# B&R Automation Studio project TD52 (part 66)

```c
    /* End of Switch: '<Root>/GasStop8' */
  }

  for (i = 0; i < 7; i++) {
    Gen2_ref_Y->out.rKengMap_P[i] = (real32_T)Gen2_ref_DWork->y_map_i[i];
  }

  Gen2_ref_Y->out.rPos_CBV2 = (real32_T)rtb_Switch_g[6];
  Gen2_ref_Y->out.rPos_CBV3 = (real32_T)rtb_Switch_g[7];
  Gen2_ref_Y->out.bAirAssistIntake = false;
  Gen2_ref_Y->out.bAirAssistExhaust = false;
  Gen2_ref_Y->out.rPos_AAV_Intake = 0.0F;
  Gen2_ref_Y->out.rPos_AAV_Exhaust = 0.0F;
  Gen2_ref_Y->out.TJ_GasO[0] = false;
  Gen2_ref_Y->out.TJ_GasO[3] = false;
  Gen2_ref_Y->out.TJ_GasO[4] = false;
  Gen2_ref_Y->out.TJ_GasM[0] = false;
  Gen2_ref_Y->out.TJ_GasM[1] = ((rtb_SumofElements -
    Gen2_ref_DWork->UnitDelay_DSTATE_dk > rtb_Gain7) &&
    (Gen2_ref_DWork->UnitDelay2_DSTATE_k - Gen2_ref_DWork->UnitDelay1_DSTATE_b >
     Gen2_ref_DWork->UnitDelay3_DSTATE_m) &&
    Gen2_ref_B->BusInput3.fdc.bActive_GasFlowStepLimit);
  Gen2_ref_Y->out.TJ_GasM[2] = ((rtb_SumofElements_l -
    Gen2_ref_DWork->UnitDelay_DSTATE_m > rtb_Sum_gb) &&
    (Gen2_ref_DWork->UnitDelay2_DSTATE_p - Gen2_ref_DWork->UnitDelay1_DSTATE_c2 >
     Gen2_ref_DWork->UnitDelay3_DSTATE_h) &&
    Gen2_ref_B->BusInput3.fdc.bActive_GasFlowStepLimit);
  Gen2_ref_Y->out.TJ_GasM[3] = false;
  Gen2_ref_Y->out.TJ_GasM[4] = false;
  Gen2_ref_Y->out.bSS = Gen2_ref_B->TON2.LogicalOperator3;

  /* Switch: '<S856>/Switch' incorporates:
   *  Constant: '<S856>/Constant2'
   *  RelationalOperator: '<S856>/Relational Operator'
   */
  if (2.2204460492503131E-16 >= rtb_Divide2_f) {
    r = 2.2204460492503131E-16;
  }

  /* End of Switch: '<S856>/Switch' */

  /* BusCreator: '<S16>/Bus Creator' incorporates:
   *  DataTypeConversion: '<S16>/Data Type Conversion20'
   *  Outport: '<Root>/out'
   *  Product: '<S13>/Product'
   */
  Gen2_ref_Y->out.rLHV_est = (real32_T)(rtb_Switch_n / r);

  /* Gain: '<S7>/W2kW' */
  r = 0.001 * rtb_Switch2_g3;

  /* BusCreator: '<Root>/Bus Creator' incorporates:
   *  BusCreator: '<S7>/Bus Creator2'
   *  DataTypeConversion: '<S7>/Data Type Conversion2'
   *  Outport: '<Root>/dbg'
   */
  Gen2_ref_Y->dbg.HLC.Gen2DbgHlcTraj.rP_Set_Delta_FSM = (real32_T)r;

  /* BusCreator generated from: '<S5>/Bus Creator' incorporates:
   *  Constant: '<S307>/Constant2'
   *  DataTypeConversion: '<S272>/Data Type Conversion'
   *  DataTypeConversion: '<S272>/Data Type Conversion1'
   *  DataTypeConversion: '<S272>/Data Type Conversion2'
   *  DataTypeConversion: '<S272>/Data Type Conversion3'
   *  DataTypeConversion: '<S272>/Data Type Conversion4'
   *  DataTypeConversion: '<S272>/Data Type Conversion5'
   *  DataTypeConversion: '<S272>/Data Type Conversion6'
   *  DataTypeConversion: '<S272>/Data Type Conversion7'
   *  DataTypeConversion: '<S272>/Data Type Conversion8'
   *  DataTypeConversion: '<S272>/Data Type Conversion9'
   *  DiscreteIntegrator: '<S307>/Discrete-Time Integrator'
   *  Sum: '<S307>/Sum4'
   */
  Gen2_ref_Y->dbg.FDC.dbgFDC_Filtering.p2s_raw = (real32_T)rtb_p2s;
  Gen2_ref_Y->dbg.FDC.dbgFDC_Filtering.p2s_1stOrd = (real32_T)
    Gen2_ref_B->sf_FILTERnodelay5.y;
  Gen2_ref_Y->dbg.FDC.dbgFDC_Filtering.p2s_2ndOrd = (real32_T)
    Gen2_ref_B->undOrderFilter3.Switch;
  Gen2_ref_Y->dbg.FDC.dbgFDC_Filtering.ne_raw = (real32_T)
    rtb_DataTypeConversion15;
  Gen2_ref_Y->dbg.FDC.dbgFDC_Filtering.ne_1stOrd = (real32_T)
    Gen2_ref_B->sf_FILTERnodelay4.y;
  Gen2_ref_Y->dbg.FDC.dbgFDC_Filtering.ne_2ndOrd = (real32_T)rtb_Switch_kr;
  Gen2_ref_Y->dbg.FDC.dbgFDC_Filtering.p2s_in = (real32_T)rtb_Switch4_p;
  Gen2_ref_Y->dbg.FDC.dbgFDC_Filtering.ne_in = (real32_T)rtb_Switch5_nn;
  Gen2_ref_Y->dbg.FDC.dbgFDC_Filtering.Ratio1stOrd = (real32_T)(1.0 -
    Gen2_ref_DWork->DiscreteTimeIntegrator_DSTATE_d);
  Gen2_ref_Y->dbg.FDC.dbgFDC_Filtering.Ratio2ndOrd = (real32_T)
    Gen2_ref_DWork->DiscreteTimeIntegrator_DSTATE_d;

  /* BusCreator generated from: '<S5>/Bus Creator' incorporates:
   *  DataTypeConversion: '<S5>/Data Type Conversion1'
   *  DataTypeConversion: '<S5>/Data Type Conversion10'
   *  DataTypeConversion: '<S5>/Data Type Conversion11'
   *  DataTypeConversion: '<S5>/Data Type Conversion2'
   *  DataTypeConversion: '<S5>/Data Type Conversion3'
   *  DataTypeConversion: '<S5>/Data Type Conversion4'
   *  DataTypeConversion: '<S5>/Data Type Conversion9'
   *  Product: '<S267>/Divide3'
   */
  Gen2_ref_Y->dbg.FDC.dbgFDC_GasArt1and2.mdot_dyn = (real32_T)rtb_Divide1_h4;
  Gen2_ref_Y->dbg.FDC.dbgFDC_GasArt1and2.mdot_set = (real32_T)rtb_SumofElements;
  Gen2_ref_Y->dbg.FDC.dbgFDC_GasArt1and2.mdot_ss = (real32_T)rtb_Product3_g;
  Gen2_ref_Y->dbg.FDC.dbgFDC_GasArt1and2.rFactCompLR = (real32_T)rtb_Switch2_l;
  Gen2_ref_Y->dbg.FDC.dbgFDC_GasArt1and2.Rgas12 = (real32_T)rtb_Divide3_n_tmp;
  Gen2_ref_Y->dbg.FDC.dbgFDC_GasArt1and2.rdpdt[0] = (real32_T)
    rtb_Switch2_gd_idx_0;
  Gen2_ref_Y->dbg.FDC.dbgFDC_GasArt1and2.rmdot_mix_dyn[0] = (real32_T)R_2inp[0];

  /* BusCreator generated from: '<S5>/Bus Creator' incorporates:
   *  DataTypeConversion: '<S5>/Data Type Conversion5'
   */
  Gen2_ref_Y->dbg.FDC.dbgFDC_GasArt3.rmdot_mix_dyn_M[0] = (real32_T)
    rtb_Divide_ab[0];

  /* BusCreator generated from: '<S5>/Bus Creator' incorporates:
   *  DataTypeConversion: '<S5>/Data Type Conversion1'
   *  DataTypeConversion: '<S5>/Data Type Conversion10'
   */
  Gen2_ref_Y->dbg.FDC.dbgFDC_GasArt1and2.rdpdt[1] = (real32_T)
    rtb_Switch2_gd_idx_1;
  Gen2_ref_Y->dbg.FDC.dbgFDC_GasArt1and2.rmdot_mix_dyn[1] = (real32_T)R_2inp[1];

  /* BusCreator generated from: '<S5>/Bus Creator' incorporates:
   *  DataTypeConversion: '<S5>/Data Type Conversion5'
   */
  Gen2_ref_Y->dbg.FDC.dbgFDC_GasArt3.rmdot_mix_dyn_M[1] = (real32_T)
    rtb_Divide_ab[1];

  /* BusCreator generated from: '<S5>/Bus Creator' incorporates:
   *  DataTypeConversion: '<S5>/Data Type Conversion1'
   *  DataTypeConversion: '<S5>/Data Type Conversion10'
   */
  Gen2_ref_Y->dbg.FDC.dbgFDC_GasArt1and2.rdpdt[2] = (real32_T)
    rtb_Switch2_gd_idx_2;
  Gen2_ref_Y->dbg.FDC.dbgFDC_GasArt1and2.rmdot_mix_dyn[2] = (real32_T)R_2inp[2];

  /* BusCreator generated from: '<S5>/Bus Creator' incorporates:
   *  DataTypeConversion: '<S5>/Data Type Conversion5'
   */
  Gen2_ref_Y->dbg.FDC.dbgFDC_GasArt3.rmdot_mix_dyn_M[2] = (real32_T)
    rtb_Divide_ab[2];

  /* BusCreator generated from: '<S5>/Bus Creator' incorporates:
   *  DataTypeConversion: '<S5>/Data Type Conversion1'
   *  DataTypeConversion: '<S5>/Data Type Conversion10'
   */
  Gen2_ref_Y->dbg.FDC.dbgFDC_GasArt1and2.rdpdt[3] = (real32_T)
    rtb_Switch2_gd_idx_3;
  Gen2_ref_Y->dbg.FDC.dbgFDC_GasArt1and2.rmdot_mix_dyn[3] = (real32_T)R_2inp[3];

  /* BusCreator generated from: '<S5>/Bus Creator' incorporates:
   *  DataTypeConversion: '<S5>/Data Type Conversion12'
   *  DataTypeConversion: '<S5>/Data Type Conversion5'
   *  DataTypeConversion: '<S5>/Data Type Conversion6'
   *  DataTypeConversion: '<S5>/Data Type Conversion7'
   *  DataTypeConversion: '<S5>/Data Type Conversion8'
   *  Product: '<S268>/Divide3'
   */
  Gen2_ref_Y->dbg.FDC.dbgFDC_GasArt3.rmdot_mix_dyn_M[3] = (real32_T)
    rtb_Divide_ab[3];
  Gen2_ref_Y->dbg.FDC.dbgFDC_GasArt3.mdot_dyn_M = (real32_T)rtb_Sum_mf;
  Gen2_ref_Y->dbg.FDC.dbgFDC_GasArt3.mdot_set_M = (real32_T)rtb_SumofElements_l;
  Gen2_ref_Y->dbg.FDC.dbgFDC_GasArt3.mdot_ss_M = (real32_T)rtb_Sum2_a1;
  Gen2_ref_Y->dbg.FDC.dbgFDC_GasArt3.Rgas3 = (real32_T)rtb_Switch_ks;

  /* BusCreator: '<S9>/Bus Creator' incorporates:
   *  DataTypeConversion: '<S9>/Data Type Conversion3'
   */
  Gen2_ref_Y->dbg.ITC.IT_off_start = 0.0F;
  Gen2_ref_Y->dbg.ITC.IT_off_island34 = 0.0F;
  Gen2_ref_Y->dbg.ITC.IT_off_island6 = (real32_T)rtb_Sum1_dh;

  /* BusCreator: '<S19>/Bus Creator' incorporates:
   *  DataTypeConversion: '<S19>/Data Type Conversion2'
   *  DataTypeConversion: '<S19>/Data Type Conversion3'
   *  DataTypeConversion: '<S19>/Data Type Conversion4'
   *  DataTypeConversion: '<S19>/Data Type Conversion5'
   */
  Gen2_ref_Y->dbg.SkipF.NskipPow = (real32_T)rtb_MinMax_n;
  Gen2_ref_Y->dbg.SkipF.NskipMax = (real32_T)rtb_RoundingFunction;
  Gen2_ref_Y->dbg.SkipF.Nskip34 = (real32_T)rtb_Product1_mqz;
  Gen2_ref_Y->dbg.SkipF.Nskip6 = (real32_T)rtb_Switch2_d1;

  /* Logic: '<S14>/Logical Operator2' */
  Gen2_ref_Y->dbg.LamLim.bInitLamOffs = !rtb_LogicalOperator5_mv;

  /* BusCreator: '<S14>/Bus Creator' incorporates:
   *  DataTypeConversion: '<S14>/Data Type Conversion'
   *  DataTypeConversion: '<S14>/Data Type Conversion10'
   *  DataTypeConversion: '<S14>/Data Type Conversion2'
   *  DataTypeConversion: '<S14>/Data Type Conversion3'
   *  DataTypeConversion: '<S14>/Data Type Conversion4'
   *  DataTypeConversion: '<S14>/Data Type Conversion5'
   *  DataTypeConversion: '<S14>/Data Type Conversion7'
   *  DataTypeConversion: '<S14>/Data Type Conversion8'
   *  DataTypeConversion: '<S14>/Data Type Conversion9'
   *  DataTypeConversion: '<S4>/Data Type Conversion28'
   */
  Gen2_ref_Y->dbg.LamLim.extOffset = Gen2_ref_B->BusInput.rOffsetLamLimit;
  Gen2_ref_Y->dbg.LamLim.AutoOffset = (real32_T)Gen2_ref_B->Filter_l.Switch;
  Gen2_ref_Y->dbg.LamLim.ScaledOffsetUpLim = (real32_T)rtb_Product1_b;
  Gen2_ref_Y->dbg.LamLim.ScaledOffsetLoLim = (real32_T)rtb_Product_l0;
  Gen2_ref_Y->dbg.LamLim.offsetUpLim = (real32_T)rtb_Sum5_j;
  Gen2_ref_Y->dbg.LamLim.offsetLoLim = (real32_T)rtb_Sum8_m;
  Gen2_ref_Y->dbg.LamLim.LamLoLim = (real32_T)rtb_Switch1_k;
  Gen2_ref_Y->dbg.LamLim.LamUpLim = (real32_T)rtb_Switch2_n5;
  Gen2_ref_Y->dbg.LamLim.LamSteadyState = (real32_T)rtb_PactOut_o;
  Gen2_ref_Y->dbg.LamLim.rLamOffsInit = (real32_T)rtb_Divide6_n;
  Gen2_ref_Y->dbg.LamLim.bPminSSadaptReached_Hys = rtb_LogicalOperator12_a;

  /* Gain: '<Root>/W2kW' */
  rtb_Sum8_m = 0.001 * rtb_Gain2_ao;

  /* S-Function (sfix_look1_dyn): '<S865>/LCRScal_CD1' */
  /* Dynamic Look-Up Table Block: '<S865>/LCRScal_CD1'
   * Input0  Data Type:  Floating Point real_T
   * Input1  Data Type:  Floating Point real_T
   * Input2  Data Type:  Floating Point real_T
   * Output0 Data Type:  Floating Point real_T
   * Lookup Method: Linear_Endpoint
   *
   */
  LookUp_real_T_real_T( &(rtb_CDSet_50),
                       &Gen2_ref_B->BusInput3.bdcWgv.rCd_vect_y[0],
                       Gen2_ref_B->BusInput3.leanox.rWG_1,
                       &Gen2_ref_B->BusInput3.bdcWgv.rCd_vect_x[0], 10U, inst);

  /* S-Function (sfix_look1_dyn): '<S865>/LCRScal_CD2' */
  /* Dynamic Look-Up Table Block: '<S865>/LCRScal_CD2'
   * Input0  Data Type:  Floating Point real_T
   * Input1  Data Type:  Floating Point real_T
   * Input2  Data Type:  Floating Point real_T
   * Output0 Data Type:  Floating Point real_T
   * Lookup Method: Linear_Endpoint
   *
   */
  LookUp_real_T_real_T( &(rtb_CDSet_100),
                       &Gen2_ref_B->BusInput3.bdcWgv.rCd_vect_y[0],
                       Gen2_ref_B->BusInput3.leanox.rWG_2,
                       &Gen2_ref_B->BusInput3.bdcWgv.rCd_vect_x[0], 10U, inst);

  /* SignalConversion generated from: '<S867>/ SFunction ' incorporates:
   *  MATLAB Function: '<S15>/LookUp Extrapolation'
   *  SignalConversion generated from: '<S15>/LCRScal_DPWG4'
   */
  rtb_TmpSignalConversionAtLoo_ht[0] = Gen2_ref_B->BusInput3.leanox.rP_1;
  rtb_TmpSignalConversionAtLoo_ht[1] = Gen2_ref_B->BusInput3.leanox.rP_2;

  /* SignalConversion generated from: '<S867>/ SFunction ' incorporates:
   *  MATLAB Function: '<S15>/LookUp Extrapolation'
   */
  rtb_TmpSignalConversionAtLook_d[0] = rtb_CDSet_50;
  rtb_TmpSignalConversionAtLook_d[1] = rtb_CDSet_100;

  /* MATLAB Function: '<S15>/LookUp Extrapolation' */
  if (rtb_TmpSignalConversionAtLoo_ht[0] == rtb_TmpSignalConversionAtLoo_ht[1])
  {
    rtb_DataTypeConversion15 = 0.0;
  } else {
    rtb_DataTypeConversion15 = (rtb_TmpSignalConversionAtLook_d[1] -
      rtb_TmpSignalConversionAtLook_d[0]) / (rtb_TmpSignalConversionAtLoo_ht[1]
      - rtb_TmpSignalConversionAtLoo_ht[0]);
    rtb_DataTypeConversion15 = (rtb_TmpSignalConversionAtLook_d[0] -
      rtb_TmpSignalConversionAtLoo_ht[0] * rtb_DataTypeConversion15) +
      rtb_DataTypeConversion15 * rtb_Sum8_m;
    if (!(rtb_DataTypeConversion15 >= 0.0)) {
      rtb_DataTypeConversion15 = 0.0;
    }

    if (!(rtb_DataTypeConversion15 <= 1.0)) {
      rtb_DataTypeConversion15 = 1.0;
    }
  }

  /* DataTypeConversion: '<S15>/Data Type Conversion' */
  r = Gen2_ref_B->BusInput.tLvrt.rWgPosFb;

  /* Gain: '<S15>/Gain' */
  rtb_Sum_e = 100.0 * r;

  /* S-Function (sfix_look1_dyn): '<S15>/LCRScal_DPWG2' */
  /* Dynamic Look-Up Table Block: '<S15>/LCRScal_DPWG2'
   * Input0  Data Type:  Floating Point real_T
   * Input1  Data Type:  Floating Point real_T
   * Input2  Data Type:  Floating Point real_T
   * Output0 Data Type:  Floating Point real_T
   * Lookup Method: Linear_Endpoint
   *
   */
  LookUp_real_T_real_T( &(rtb_Sum_mf), &Gen2_ref_B->BusInput3.bdcWgv.rCd_vect_y
                       [0], rtb_Sum_e, &Gen2_ref_B->BusInput3.bdcWgv.rCd_vect_x
                       [0], 10U, inst);

  /* BusCreator: '<Root>/Bus Creator1' incorporates:
   *  DataTypeConversion: '<Root>/Data Type Conversion4'
   */
  Gen2_ref_Y->dbg.LxWgvCmp.CDAct = (real32_T)rtb_Sum_mf;

  /* Math: '<S868>/Math Function' */
  r = Gen2_ref_B->BusInput3.bdcWgv.rDref * Gen2_ref_B->BusInput3.bdcWgv.rDref;

  /* Abs: '<S871>/Abs' */
  rtb_Divide2_f = fabs(Gen2_ref_B->BusInput3.eng.rVol_Hub_Eng);

  /* Switch: '<S871>/Switch' incorporates:
   *  Constant: '<S871>/Constant2'
   *  RelationalOperator: '<S871>/Relational Operator'
   */
  if (2.2204460492503131E-16 >= rtb_Divide2_f) {
    rtb_Divide2_f = 2.2204460492503131E-16;
  } else {
    rtb_Divide2_f = Gen2_ref_B->BusInput3.eng.rVol_Hub_Eng;
  }

  /* End of Switch: '<S871>/Switch' */

  /* Product: '<S868>/Divide' incorporates:
   *  Constant: '<S868>/Constant'
   *  Sum: '<S15>/Add1'
   */
  rtb_Sum_mf = (rtb_DataTypeConversion15 - rtb_Sum_mf) * r * 0.78539816339744828
    * Gen2_ref_B->BusInput3.eng.rNum_WGV / rtb_Divide2_f;

  /* SignalConversion generated from: '<S15>/LCRScal_DPWG4' */
  rtb_TmpSignalConversionAtLook_d[0] = rtb_TmpSignalConversionAtLoo_ht[0];
  rtb_TmpSignalConversionAtLook_d[1] = rtb_TmpSignalConversionAtLoo_ht[1];

  /* S-Function (sfix_look1_dyn): '<S15>/LCRScal_DPWG3' */
  /* Dynamic Look-Up Table Block: '<S15>/LCRScal_DPWG3'
   * Input0  Data Type:  Floating Point real_T
   * Input1  Data Type:  Floating Point real_T
   * Input2  Data Type:  Floating Point real_T
   * Output0 Data Type:  Floating Point real_T
   * Lookup Method: Linear_Endpoint
   *
   */
  LookUp_real_T_real_T( &(r), &Gen2_ref_B->BusInput3.leanox.Comp_WG_1_y[0],
                       rtb_Sum_mf, &Gen2_ref_B->BusInput3.leanox.Comp_WG_1_x[0],
                       9U, inst);

  /* S-Function (sfix_look1_dyn): '<S15>/LCRScal_DPWG1' */
  /* Dynamic Look-Up Table Block: '<S15>/LCRScal_DPWG1'
   * Input0  Data Type:  Floating Point real_T
   * Input1  Data Type:  Floating Point real_T
   * Input2  Data Type:  Floating Point real_T
   * Output0 Data Type:  Floating Point real_T
   * Lookup Method: Linear_Endpoint
   *
   */
  LookUp_real_T_real_T( &(rtb_Divide2_f),
                       &Gen2_ref_B->BusInput3.leanox.Comp_WG_2_y[0], rtb_Sum_mf,
                       &Gen2_ref_B->BusInput3.leanox.Comp_WG_2_x[0], 9U, inst);

  /* SignalConversion generated from: '<S15>/LCRScal_DPWG4' */
  rtb_TmpSignalConversionAtLoo_ht[0] = r;
  rtb_TmpSignalConversionAtLoo_ht[1] = rtb_Divide2_f;

  /* S-Function (sfix_look1_dyn): '<S15>/LCRScal_DPWG4' */
  /* Dynamic Look-Up Table Block: '<S15>/LCRScal_DPWG4'
   * Input0  Data Type:  Floating Point real_T
   * Input1  Data Type:  Floating Point real_T
   * Input2  Data Type:  Floating Point real_T
   * Output0 Data Type:  Floating Point real_T
   * Lookup Method: Linear_Endpoint
   *
   */
  LookUp_real_T_real_T( &(r), &rtb_TmpSignalConversionAtLoo_ht[0], rtb_Sum8_m,
                       &rtb_TmpSignalConversionAtLook_d[0], 1U, inst);

  /* BusCreator: '<Root>/Bus Creator1' incorporates:
   *  DataTypeConversion: '<Root>/Data Type Conversion3'
   *  DataTypeConversion: '<Root>/Data Type Conversion5'
   *  DataTypeConversion: '<Root>/Data Type Conversion6'
   *  DataTypeConversion: '<Root>/Data Type Conversion8'
   *  Delay: '<S15>/Resettable Delay'
   */
  Gen2_ref_Y->dbg.LxWgvCmp.CDSet = (real32_T)rtb_DataTypeConversion15;
  Gen2_ref_Y->dbg.LxWgvCmp.DeltaCD_aux = (real32_T)rtb_Sum_mf;
  Gen2_ref_Y->dbg.LxWgvCmp.DeltaP2s_set = (real32_T)r;
  Gen2_ref_Y->dbg.LxWgvCmp.DeltaP2s_Comp_WGV = (real32_T)
    Gen2_ref_DWork->ResettableDelay_DSTATE;

  /* BusCreator: '<S6>/Bus Creator' incorporates:
   *  Delay: '<Root>/Delay6'
   */
  Gen2_ref_Y->dbg.GQC.bActGasQualImprov = rtb_bActGasQualImprov;
  Gen2_ref_Y->dbg.GQC.bDetSatLambda = rtb_LogicalOperator2_fy;
  Gen2_ref_Y->dbg.GQC.bDetKnock = rtb_Switch2_jv;
  Gen2_ref_Y->dbg.GQC.bDetSatActuators = Gen2_ref_DWork->Delay6_DSTATE;
  Gen2_ref_Y->dbg.GQC.bMisfDet = rtb_Switch4_mu;

  /* BusCreator: '<Root>/Bus Creator' incorporates:
   *  BusCreator: '<S427>/Bus Creator5'
   *  BusCreator: '<S429>/Bus Creator'
   *  DataTypeConversion: '<S418>/Data Type Conversion10'
   *  DataTypeConversion: '<S418>/Data Type Conversion11'
   *  DataTypeConversion: '<S418>/Data Type Conversion12'
   *  DataTypeConversion: '<S418>/Data Type Conversion13'
   *  DataTypeConversion: '<S427>/Data Type Conversion'
   *  DataTypeConversion: '<S427>/Data Type Conversion1'
   *  DataTypeConversion: '<S427>/Data Type Conversion2'
   *  DataTypeConversion: '<S427>/Data Type Conversion3'
   *  DataTypeConversion: '<S427>/Data Type Conversion4'
   *  DataTypeConversion: '<S429>/Data Type Conversion1'
   *  DataTypeConversion: '<S429>/Data Type Conversion4'
   *  DataTypeConversion: '<S429>/Data Type Conversion5'
   *  DataTypeConversion: '<S432>/Data Type Conversion1'
   *  DataTypeConversion: '<S432>/Data Type Conversion10'
   *  DataTypeConversion: '<S432>/Data Type Conversion11'
   *  DataTypeConversion: '<S432>/Data Type Conversion2'
   *  DataTypeConversion: '<S432>/Data Type Conversion3'
   *  DataTypeConversion: '<S432>/Data Type Conversion4'
   *  DataTypeConversion: '<S432>/Data Type Conversion5'
   *  DataTypeConversion: '<S432>/Data Type Conversion6'
   *  DataTypeConversion: '<S581>/Data Type Conversion6'
   *  Outport: '<Root>/dbg'
   *  Quantizer: '<S581>/Quantizer1'
   */
  Gen2_ref_Y->dbg.HLCi.FF.rPest_FF = (real32_T)rtb_Switch_bs;
  Gen2_ref_Y->dbg.HLCi.FF.rP2s_FF = (real32_T)rtb_mbar2pa_g;
  Gen2_ref_Y->dbg.HLCi.FF.P_est_vFilt = (real32_T)rtb_Switch2_gs;
  Gen2_ref_Y->dbg.HLCi.FF.LineVol_nPower = (real32_T)rtb_Switch_iy;
  Gen2_ref_Y->dbg.HLCi.FF.LineVol_vPower = (real32_T)rtb_rKK2_k;
  Gen2_ref_Y->dbg.HLCi.FF.rFactLSL = (real32_T)rtb_Sum1_jz;
  Gen2_ref_Y->dbg.HLCi.FF.rLSLff_p = (real32_T)rtb_Divide_kp;
  Gen2_ref_Y->dbg.HLCi.FF.rLSLff_d = (real32_T)rtb_Divide2_a;
  Gen2_ref_Y->dbg.HLCi.LR.bLR_GasStop = rtb_TOF_IN;
  Gen2_ref_Y->dbg.HLCi.LR.bIgnOff = rtb_bCBV_min;
  Gen2_ref_Y->dbg.HLCi.LR.bLR_ActSat_CBV =
    Gen2_ref_B->TP_ActSat_CBV.LogicalOperator1;
  Gen2_ref_Y->dbg.HLCi.LR.bLR_ActSat_TV =
    Gen2_ref_B->TP_ActSat_TV.LogicalOperator1;
  Gen2_ref_Y->dbg.HLCi.LR.bLR_IGN_Retard_Trig = rtb_RelationalOperator2_j;
  Gen2_ref_Y->dbg.HLCi.LR.rP_Rot_Corr_Norm = (real32_T)rtb_Saturation;
  Gen2_ref_Y->dbg.HLCi.LR.IGN_retard_interpol = (real32_T)rtb_Switch2_jq;
  Gen2_ref_Y->dbg.HLCi.LR.IGN_retard_active = (real32_T)rtb_Divide4_d;
  Gen2_ref_Y->dbg.HLCi.LR.delta_IGN_Retard = (real32_T)rtb_MinMax_a;
  Gen2_ref_Y->dbg.HLCi.LR.rFactCompLR = (real32_T)rtb_Switch2_l;
  Gen2_ref_Y->dbg.HLCi.LR.bLR_SatActuators = rtb_LogicalOperator3_gq;
  Gen2_ref_Y->dbg.HLCi.Prot.omega = (real32_T)rtb_Gain;
  Gen2_ref_Y->dbg.HLCi.Prot.omega_filt = (real32_T)rtb_Switch_eu;
  Gen2_ref_Y->dbg.HLCi.Prot.omega_dot = (real32_T)rtb_Switch1_mm;
  Gen2_ref_Y->dbg.HLCi.Prot.rProt = (real32_T)rtb_Gain1_fr;
  Gen2_ref_Y->dbg.HLCi.SkipF.rSkipfire_PI = (real32_T)rtb_Switch2_ba;
  Gen2_ref_Y->dbg.HLCi.SkipF.rLam_skip = (real32_T)rtb_Switch_fi;
  Gen2_ref_Y->dbg.HLCi.SkipF.bDemand_Skip = rtb_LogicalOperator1_ja;
  Gen2_ref_Y->dbg.HLCi.SkipF.rSkip_level = (real32_T)rtb_rSkip_level;
  Gen2_ref_Y->dbg.HLCi.SkipF.rSkipfire = (real32_T)rtb_Divide1_f1_tmp;
  Gen2_ref_Y->dbg.HLCi.SkipF.bSkip_pulse_on = rtb_LogicalOperator1_pa;

  /* Switch: '<S429>/Switch1' incorporates:
   *  BusCreator: '<Root>/Bus Creator'
   *  DataTypeConversion: '<S429>/Data Type Conversion2'
   *  Outport: '<Root>/dbg'
   */
  Gen2_ref_Y->dbg.HLCi.SkipF.rN_diff = (real32_T)rtb_Divide_mr_tmp;

  /* BusCreator: '<Root>/Bus Creator' incorporates:
   *  BusCreator: '<S1>/Bus Creator2'
   *  BusCreator: '<S23>/Bus Creator1'
   *  BusCreator: '<S389>/Bus Creator1'
   *  BusCreator: '<S431>/Bus Creator'
   *  BusCreator: '<S7>/Bus Creator2'
   *  DataTypeConversion: '<S12>/Data Type Conversion1'
   *  DataTypeConversion: '<S1>/Data Type Conversion'
   *  DataTypeConversion: '<S1>/Data Type Conversion1'
   *  DataTypeConversion: '<S1>/Data Type Conversion10'
   *  DataTypeConversion: '<S1>/Data Type Conversion16'
   *  DataTypeConversion: '<S1>/Data Type Conversion17'
   *  DataTypeConversion: '<S1>/Data Type Conversion18'
   *  DataTypeConversion: '<S1>/Data Type Conversion2'
   *  DataTypeConversion: '<S1>/Data Type Conversion22'
   *  DataTypeConversion: '<S1>/Data Type Conversion23'
   *  DataTypeConversion: '<S1>/Data Type Conversion24'
   *  DataTypeConversion: '<S1>/Data Type Conversion3'
   *  DataTypeConversion: '<S1>/Data Type Conversion4'
   *  DataTypeConversion: '<S1>/Data Type Conversion5'
   *  DataTypeConversion: '<S1>/Data Type Conversion6'
   *  DataTypeConversion: '<S1>/Data Type Conversion8'
   *  DataTypeConversion: '<S23>/Data Type Conversion'
   *  DataTypeConversion: '<S23>/Data Type Conversion1'
   *  DataTypeConversion: '<S23>/Data Type Conversion2'
   *  DataTypeConversion: '<S23>/Data Type Conversion3'
   *  DataTypeConversion: '<S23>/Data Type Conversion4'
   *  DataTypeConversion: '<S23>/Data Type Conversion6'
   *  DataTypeConversion: '<S23>/Data Type Conversion7'
   *  DataTypeConversion: '<S26>/Data Type Conversion'
   *  DataTypeConversion: '<S26>/Data Type Conversion2'
   *  DataTypeConversion: '<S26>/Data Type Conversion3'
   *  DataTypeConversion: '<S26>/Data Type Conversion4'
   *  DataTypeConversion: '<S26>/Data Type Conversion5'
   *  DataTypeConversion: '<S26>/Data Type Conversion7'
   *  DataTypeConversion: '<S379>/Data Type Conversion10'
   *  DataTypeConversion: '<S379>/Data Type Conversion3'
   *  DataTypeConversion: '<S379>/Data Type Conversion5'
   *  DataTypeConversion: '<S379>/Data Type Conversion8'
   *  DataTypeConversion: '<S389>/Data Type Conversion3'
   *  DataTypeConversion: '<S389>/Data Type Conversion6'
   *  DataTypeConversion: '<S389>/Data Type Conversion8'
   *  DataTypeConversion: '<S431>/Data Type Conversion1'
   *  DataTypeConversion: '<S431>/Data Type Conversion10'
   *  DataTypeConversion: '<S431>/Data Type Conversion11'
   *  DataTypeConversion: '<S431>/Data Type Conversion12'
   *  DataTypeConversion: '<S431>/Data Type Conversion13'
   *  DataTypeConversion: '<S431>/Data Type Conversion14'
   *  DataTypeConversion: '<S431>/Data Type Conversion15'
   *  DataTypeConversion: '<S431>/Data Type Conversion16'
   *  DataTypeConversion: '<S431>/Data Type Conversion17'
   *  DataTypeConversion: '<S431>/Data Type Conversion18'
   *  DataTypeConversion: '<S431>/Data Type Conversion19'
   *  DataTypeConversion: '<S431>/Data Type Conversion2'
   *  DataTypeConversion: '<S431>/Data Type Conversion20'
   *  DataTypeConversion: '<S431>/Data Type Conversion21'
   *  DataTypeConversion: '<S431>/Data Type Conversion22'
   *  DataTypeConversion: '<S431>/Data Type Conversion23'
   *  DataTypeConversion: '<S431>/Data Type Conversion24'
   *  DataTypeConversion: '<S431>/Data Type Conversion25'
   *  DataTypeConversion: '<S431>/Data Type Conversion26'
   *  DataTypeConversion: '<S431>/Data Type Conversion27'
   *  DataTypeConversion: '<S431>/Data Type Conversion3'
   *  DataTypeConversion: '<S431>/Data Type Conversion4'
   *  DataTypeConversion: '<S431>/Data Type Conversion5'
   *  DataTypeConversion: '<S431>/Data Type Conversion6'
   *  DataTypeConversion: '<S431>/Data Type Conversion7'
   *  DataTypeConversion: '<S431>/Data Type Conversion8'
   *  DataTypeConversion: '<S431>/Data Type Conversion9'
   *  DataTypeConversion: '<S43>/Data Type Conversion1'
   *  DataTypeConversion: '<S43>/Data Type Conversion24'
   *  DataTypeConversion: '<S43>/Data Type Conversion25'
   *  DataTypeConversion: '<S43>/Data Type Conversion3'
   *  DataTypeConversion: '<S45>/Data Type Conversion'
   *  DataTypeConversion: '<S45>/Data Type Conversion2'
   *  DataTypeConversion: '<S45>/Data Type Conversion3'
   *  DataTypeConversion: '<S45>/Data Type Conversion4'
   *  DataTypeConversion: '<S45>/Data Type Conversion7'
   *  DataTypeConversion: '<S4>/Data Type Conversion29'
   *  DataTypeConversion: '<S78>/Data Type Conversion1'
   *  DataTypeConversion: '<S78>/Data Type Conversion10'
   *  DataTypeConversion: '<S78>/Data Type Conversion2'
   *  DataTypeConversion: '<S78>/Data Type Conversion3'
   *  DataTypeConversion: '<S78>/Data Type Conversion4'
   *  DataTypeConversion: '<S78>/Data Type Conversion5'
   *  DataTypeConversion: '<S78>/Data Type Conversion7'
   *  DataTypeConversion: '<S78>/Data Type Conversion8'
   *  DataTypeConversion: '<S78>/Data Type Conversion9'
   *  DataTypeConversion: '<S7>/Data Type Conversion1'
   *  DiscreteIntegrator: '<S26>/Discrete-Time Integrator'
   *  DiscreteIntegrator: '<S45>/Discrete-Time Integrator1'
   *  DiscreteIntegrator: '<S62>/Discrete-Time Integrator'
   *  DiscreteIntegrator: '<S748>/Discrete-Time Integrator4'
   *  Gain: '<S431>/Gain1'
   *  Gain: '<S7>/Pa2bar'
   *  Logic: '<S45>/Logical Operator'
   *  MATLAB Function: '<S431>/LQR Controller 3states'
   *  Outport: '<Root>/dbg'
   *  SignalConversion generated from: '<S627>/ SFunction '
   *  Sum: '<S641>/Sum2'
   *  Sum: '<S641>/Sum6'
   */
  Gen2_ref_Y->dbg.HLCi.LQR.x_ref[0] = (real32_T)rtb_Saturation6;
  Gen2_ref_Y->dbg.HLCi.LQR.x_ref[1] = (real32_T)rtb_Abs;
  Gen2_ref_Y->dbg.HLCi.LQR.x_ref[2] = (real32_T)rtb_Switch2_c4;
  Gen2_ref_Y->dbg.HLCi.LQR.x_sp[0] = (real32_T)rtb_Sum1_l;
  Gen2_ref_Y->dbg.HLCi.LQR.x_sp[1] = (real32_T)rtb_Sum2_a_tmp;
  Gen2_ref_Y->dbg.HLCi.LQR.x_sp[2] = (real32_T)rtb_Sum6_o_tmp;
  Gen2_ref_Y->dbg.HLCi.LQR.x_k[0] = (real32_T)rtb_Gain1_f_tmp;
  Gen2_ref_Y->dbg.HLCi.LQR.x_k[1] = (real32_T)rtb_Gain3;
  Gen2_ref_Y->dbg.HLCi.LQR.x_k[2] = (real32_T)Gen2_ref_B->Filter_bd.Switch;
  Gen2_ref_Y->dbg.HLCi.LQR.u_k[0] = (real32_T)rtb_Product_m[0];
  Gen2_ref_Y->dbg.HLCi.LQR.u_k[1] = (real32_T)rtb_Product_m[1];
  Gen2_ref_Y->dbg.HLCi.LQR.u_k[2] = (real32_T)rtb_Product_m[2];
  Gen2_ref_Y->dbg.HLCi.LQR.u_k[3] = (real32_T)rtb_Product_m[3];
  Gen2_ref_Y->dbg.HLCi.LQR.x_dist1_map = (real32_T)rtb_Gain1_o;
  Gen2_ref_Y->dbg.HLCi.LQR.x_KF[0] = (real32_T)rtb_x_KF_out_idx_0;
  Gen2_ref_Y->dbg.HLCi.LQR.x_dist_KF[0] = (real32_T)rtb_Switch1_cl[0];
  Gen2_ref_Y->dbg.HLCi.LQR.x_sp_KF[0] = (real32_T)rtb_x_sp_KF_idx_0;
  Gen2_ref_Y->dbg.HLCi.LQR.x_KF[1] = (real32_T)rtb_x_KF_out_idx_1;
  Gen2_ref_Y->dbg.HLCi.LQR.x_dist_KF[1] = (real32_T)rtb_Switch1_cl[1];
  Gen2_ref_Y->dbg.HLCi.LQR.x_sp_KF[1] = (real32_T)rtb_x_sp_KF_idx_1;
  Gen2_ref_Y->dbg.HLCi.LQR.x_KF[2] = (real32_T)rtb_x_KF_out_idx_2;
  Gen2_ref_Y->dbg.HLCi.LQR.x_dist_KF[2] = (real32_T)rtb_Switch1_cl[2];
  Gen2_ref_Y->dbg.HLCi.LQR.x_sp_KF[2] = (real32_T)rtb_x_sp_KF_idx_2;
  Gen2_ref_Y->dbg.HLCi.LQR.u_sp_KF[0] = (real32_T)rtb_u_sp_KF[0];
  Gen2_ref_Y->dbg.HLCi.LQR.u_sp_KF[1] = (real32_T)rtb_u_sp_KF[1];
  Gen2_ref_Y->dbg.HLCi.LQR.err_KF[0] = (real32_T)rtb_err_KF[0];
  Gen2_ref_Y->dbg.HLCi.LQR.err_KF[1] = (real32_T)rtb_err_KF[1];
  Gen2_ref_Y->dbg.HLCi.LQR.err_KF[2] = (real32_T)rtb_err_KF[2];
  for (i = 0; i < 18; i++) {
    Gen2_ref_Y->dbg.HLCi.LQR.K_KF[i] = (real32_T)rtb_K_KF_out[i];
  }

  for (i = 0; i < 36; i++) {
    Gen2_ref_Y->dbg.HLCi.LQR.P_KF[i] = (real32_T)Gen2_ref_DWork->P_KF[i];
  }

  Gen2_ref_Y->dbg.HLCi.LQR.err_cont[0] = (real32_T)rtb_err_cont[0];
  Gen2_ref_Y->dbg.HLCi.LQR.err_cont[1] = (real32_T)rtb_err_cont[1];
  Gen2_ref_Y->dbg.HLCi.LQR.err_cont[2] = (real32_T)rtb_err_cont[2];
  Gen2_ref_Y->dbg.HLCi.LQR.Ke_calc = (real32_T)rtb_Switch_nb;
  Gen2_ref_Y->dbg.HLCi.LQR.Ke = (real32_T)rtb_Product_o;
  Gen2_ref_Y->dbg.HLCi.LQR.Ke0 = (real32_T)rtb_VariableIntegerDelay;
  Gen2_ref_Y->dbg.HLCi.LQR.eOmRef = (real32_T)rtb_Switch_dhr;
  Gen2_ref_Y->dbg.HLCi.LQR.bTrigDPr_limit = rtb_Act;
  Gen2_ref_Y->dbg.HLCi.LQR.bOutOfNWindow = rtb_LogicalOperator4_go;
  Gen2_ref_Y->dbg.HLCi.LQR.omega_dot = (real32_T)((rtb_Product_o / (y_map_tmp_0 *
    rtb_Sum1_idx_2 + 1.0) * y_map_tmp * (rtb_Product_m[2] *
    Gen2_ref_B->BusInput3.SpeedCtrl.rK_it2_iLQR + 1.0) - rtb_Divide_i1) * (1.0 /
    rtb_TmpSignalConversionAtSFunct[3]));
  Gen2_ref_Y->dbg.HLCi.LQR.bLamSat = rtb_LogicalOperator2_ov;
  for (i = 0; i < 9; i++) {
    Gen2_ref_Y->dbg.HLCi.LQR.Phi[i] = (real32_T)rtb_Phi_OUT[i];
  }

  Gen2_ref_Y->dbg.HLCi.LQR.x_k_pred[0] = (real32_T)
    rtb_TmpSignalConversionAtSFun_g[0];
  Gen2_ref_Y->dbg.HLCi.LQR.x_k_pred[1] = (real32_T)
    rtb_TmpSignalConversionAtSFun_g[1];
  Gen2_ref_Y->dbg.HLCi.LQR.x_k_pred[2] = (real32_T)
    rtb_TmpSignalConversionAtSFun_g[2];
  for (i = 0; i < 12; i++) {
    Gen2_ref_Y->dbg.HLCi.LQR.H[i] = (real32_T)rtb_H_OUT[i];
    Gen2_ref_Y->dbg.HLCi.LQR.K_LQR[i] = (real32_T)rtb_K_LQR[i];
  }

  for (i = 0; i < 9; i++) {
    Gen2_ref_Y->dbg.HLCi.LQR.P_LQR[i] = (real32_T)Gen2_ref_DWork->P[i];
  }

  Gen2_ref_Y->dbg.HLCi.LQR.Ke_act_map = (real32_T)rtb_Switch1_ep;
  Gen2_ref_Y->dbg.HLCi.LQR.bAdaptReleased = rtb_RelationalOperator_ok;
  Gen2_ref_Y->dbg.HLCi.LQR.bResKeEst = rtb_Switch2_ij;
  Gen2_ref_Y->dbg.HLCi.LQR.bKeEstTransDet = rtb_Switch3_of;
  Gen2_ref_Y->dbg.HLCi.LQR.Ke_est = (real32_T)Gen2_ref_B->Filter1_o.Switch;
  Gen2_ref_Y->dbg.HLCi.LQR.delta_IT_Acc = (real32_T)rtb_Product4_d;
  Gen2_ref_Y->dbg.HLCi.LQR.dPr_P2s_RefSatLam = (real32_T)
    Gen2_ref_DWork->DiscreteTimeIntegrator4_DSTATE;
  Gen2_ref_Y->dbg.HLC.Gen2DbgHlcTraj.rp2s_leanox = (real32_T)(1.0E-5 *
    rtb_Pa2bar_k);

  /* Outputs for Atomic SubSystem: '<S342>/PID_Power' */
  Gen2_ref_Y->dbg.HLC.BGen2DbgHlcPowCtrl.ff = (real32_T)rtb_Switch_e3;
  Gen2_ref_Y->dbg.HLC.BGen2DbgHlcPowCtrl.ud = (real32_T)rtb_Divide3_p;
  Gen2_ref_Y->dbg.HLC.BGen2DbgHlcPowCtrl.aw_ext = (real32_T)rtb_Switch8;

  /* End of Outputs for SubSystem: '<S342>/PID_Power' */
  Gen2_ref_Y->dbg.HLC.BGen2DbgHlcPowCtrl.aw_aux =
    Gen2_ref_B->BusInput.rAW_EGT_ext;

  /* Outputs for Atomic SubSystem: '<S342>/PID_Power' */
  Gen2_ref_Y->dbg.HLC.BGen2DbgHlcPowCtrl.u = (real32_T)rtb_Switch2_jw;

  /* End of Outputs for SubSystem: '<S342>/PID_Power' */

  /* Outputs for Atomic SubSystem: '<S343>/PID_Power' */
  Gen2_ref_Y->dbg.HLC.dbgHLCPowCtrlGQC.ff = 0.0F;

  /* End of Outputs for SubSystem: '<S343>/PID_Power' */
  Gen2_ref_Y->dbg.HLC.dbgHLCPowCtrlGQC.ui = rtb_BusCreator1_h_ui;

  /* Outputs for Atomic SubSystem: '<S343>/PID_Power' */
  Gen2_ref_Y->dbg.HLC.dbgHLCPowCtrlGQC.ud = (real32_T)rtb_Divide3_d;
  Gen2_ref_Y->dbg.HLC.dbgHLCPowCtrlGQC.aw_ext = 0.0F;
  Gen2_ref_Y->dbg.HLC.dbgHLCPowCtrlGQC.aw_aux = (real32_T)rtb_Product1;
  Gen2_ref_Y->dbg.HLC.dbgHLCPowCtrlGQC.u = (real32_T)
    Gen2_ref_B->sf_MATLABFunction1_ep.LamOut;

  /* End of Outputs for SubSystem: '<S343>/PID_Power' */
  Gen2_ref_Y->dbg.BDC.Misc.PI_tv = (real32_T)rtb_Divide_br;
  Gen2_ref_Y->dbg.BDC.Misc.PI_LP = (real32_T)rtb_Divide2;
  Gen2_ref_Y->dbg.BDC.Misc.PI_HP = (real32_T)rtb_Divide1_fn;
  Gen2_ref_Y->dbg.BDC.Misc.PI_total = (real32_T)rtb_Divide3_a0;
  Gen2_ref_Y->dbg.BDC.tv.ff = (real32_T)
    Gen2_ref_B->Inverse_Linearization1.LCRScal_Lam_EOT1;
  Gen2_ref_Y->dbg.BDC.tv.up = (real32_T)rtb_Product4;
  Gen2_ref_Y->dbg.BDC.tv.ui = (real32_T)
    Gen2_ref_DWork->DiscreteTimeIntegrator1_DSTAT_n;
  Gen2_ref_Y->dbg.BDC.tv.uaw = (real32_T)rtb_Switch2_oou;
  Gen2_ref_Y->dbg.BDC.tv.i0 = (real32_T)rtb_Switch1_d2;
  Gen2_ref_Y->dbg.BDC.tv.bTVCtrl_ON = !rtb_i_reset;
  Gen2_ref_Y->dbg.BDC.cbv.ff_cbv = (real32_T)rtb_Saturation1_i;
  Gen2_ref_Y->dbg.BDC.cbv.ff_cbv_unsat = (real32_T)rtb_Sum1_lo;
  Gen2_ref_Y->dbg.BDC.cbv.up_cbv = (real32_T)rtb_up;
  Gen2_ref_Y->dbg.BDC.cbv.ui_cbv = (real32_T)
    Gen2_ref_DWork->DiscreteTimeIntegrator_DSTAT_ja;
  Gen2_ref_Y->dbg.BDC.cbv.uaw_cbv = (real32_T)FILT_IN;
  Gen2_ref_Y->dbg.BDC.cbv.i0_cbv = (real32_T)rtb_Add2_h;
  Gen2_ref_Y->dbg.BDC.SP.rCBV_Min = (real32_T)rtb_Switch2_a;
  Gen2_ref_Y->dbg.BDC.SP.rTV_Min = (real32_T)rtb_Switch_e;
  Gen2_ref_Y->dbg.BDC.SP.rMdot_mixture_cyl = (real32_T)rtb_MassFlowCalc;
  Gen2_ref_Y->dbg.BDC.SP.rPrR_TC_Surge = (real32_T)rtb_Saturation_gh;
  Gen2_ref_Y->dbg.BDC.MP.u = (real32_T)rtb_Sum11;
  Gen2_ref_Y->dbg.BDC.MP.u_ff = (real32_T)rtb_MinMax1_h;
  Gen2_ref_Y->dbg.BDC.MP.u0 = (real32_T)rtb_Sum7_l5;
  Gen2_ref_Y->dbg.BDC.MP.u0_ff = (real32_T)rtb_MinMax1_g;
  Gen2_ref_Y->dbg.BDC.MP.TVdp = (real32_T)rtb_Product2;
  Gen2_ref_Y->dbg.BDC.MP.offset = (real32_T)
    Gen2_ref_DWork->DiscreteTimeIntegrator_DSTATE_a;
  Gen2_ref_Y->dbg.BDC.MP.offset_in = (real32_T)rtb_Gain_kl;
  Gen2_ref_Y->dbg.BDC.RL.RLp2s_d = (real32_T)rtb_p1LP;
  Gen2_ref_Y->dbg.BDC.RL.RLp2s_d_ff = (real32_T)rtb_p1HP;
  Gen2_ref_Y->dbg.BDC.RL.RLp2s_d_ff_z = (real32_T)rtb_VariableIntegerDelay_b;
  Gen2_ref_Y->dbg.BDC.RL.RLact = (real32_T)rtb_MinMax3;
  Gen2_ref_Y->dbg.BDC.RL.RL = (real32_T)rtb_MinMax_mf;
  Gen2_ref_Y->dbg.BDC.RL.Rlrequ = (real32_T)rtb_Divide_kt;
  Gen2_ref_Y->dbg.BDC.RL.RLp2s_d_RL = (real32_T)rtb_p2HP;
  Gen2_ref_Y->dbg.BDC.RL.RLp2s_d_ff_RL = (real32_T)rtb_Sum5_iu;
  Gen2_ref_Y->dbg.BDC.RL.Rlreset = rtb_LogicalOperator3_ja;
  Gen2_ref_Y->dbg.BDC.traj.ref_P2_FF_CBV = rtb_Switch2_h1;
  Gen2_ref_Y->dbg.BDC.traj.ref_P2s_FF = rtb_Switch2_lu;
  Gen2_ref_Y->dbg.BDC.traj.ref_P2_FF = rtb_BusCreator1_ref_P2_FF;
  Gen2_ref_Y->dbg.BDC.traj.ref_P2s_FB_TV = rtb_BusCreator1_ref_P2s_FB_TV;
  Gen2_ref_Y->dbg.BDC.traj.ref_P2_FB_CBV = rtb_BusCreator1_ref_P2_FB_CBV;
  Gen2_ref_Y->dbg.BDC.traj.ref_P2s_FF_TV = rtb_Switch2_jf;
  Gen2_ref_Y->dbg.BDC.traj.d_dt_ref_P2s_FF_TV = Gen2_ref_B->Filter2.Switch1;
  Gen2_ref_Y->dbg.BDC.traj.d_dt_ref_P2_FF_CBV = Gen2_ref_B->Filter1.Switch1;
  Gen2_ref_Y->dbg.BDC.traj.d_dt_ref_P2s_FF = Gen2_ref_B->Filter4.Switch1;
  Gen2_ref_Y->dbg.BDC.FF.me = (real32_T)rtb_dm_e;
  Gen2_ref_Y->dbg.BDC.FF.me_d = (real32_T)Gen2_ref_B->sf_enginemassflow.dm_e;
  Gen2_ref_Y->dbg.BDC.FF.me_cbv_d = (real32_T)rtb_Abs_n;
  Gen2_ref_Y->dbg.BDC.FF.TV_me_d = (real32_T)rtb_Divide_n0;
  Gen2_ref_Y->dbg.BDC.FF.wg_me = (real32_T)Gen2_ref_B->sf_enginemassflow1_e.dm_e;
  Gen2_ref_Y->dbg.BDC.FF.wg_me_d = (real32_T)
    Gen2_ref_B->sf_enginemassflow_h.dm_e;
  Gen2_ref_Y->dbg.BDC.FF.wg_m_d = (real32_T)rtb_Saturation_cx;
  Gen2_ref_Y->dbg.BDC.FF.u_ff_cbv = (real32_T)rtb_Sum1_lo;
  Gen2_ref_Y->dbg.BDC.FF.dbg_cbvTracking_PI = (real32_T)rtb_Sum3_hx;
  Gen2_ref_Y->dbg.BDC.FF.dbg_cbvTracking_P = (real32_T)rtb_Divide1_k;
  Gen2_ref_Y->dbg.BDC.FF.dbg_cbvTracking_I = (real32_T)
    rtb_DiscreteTimeIntegrator_g3;
  Gen2_ref_Y->dbg.KeEstNetP.KeEstNetP = (real32_T)Gen2_ref_B->Filter1_n.Switch;

  /* S-Function (bur_bus_out): '<Root>/Bus Output' incorporates:
   *  Outport: '<Root>/dbg'
   */
  inst->dbgOut = Gen2_ref_Y->dbg;

  /* S-Function (bur_bus_out): '<Root>/Bus Output1' incorporates:
   *  Outport: '<Root>/out'
   */
  inst->OUT = Gen2_ref_Y->out;

  /* S-Function (bur_in): '<Root>/Input1' */
  Gen2_ref_B->Input1 = inst->rLam_BrakeEffEst;

  /* Outputs for Atomic SubSystem: '<Root>/brake eff estimate' */
  /* Gain: '<S21>/Gain' */
  rtb_Sum_mf = 0.10471975511965977 * Gen2_ref_B->BusInput3.eng.rN_Nom;

  /* Product: '<S21>/Divide' */
  rtb_Sum_mf = Gen2_ref_B->BusInput3.eng.rVol_Hub_Eng * rtb_Sum1_idx_3 *
    rtb_Sum_mf * rtb_etaVolConst_lt * Gen2_ref_B->p2s_filt.Switch;

  /* Product: '<S21>/Divide3' */
  rtb_Divide2_f = Gen2_ref_B->Input1 * rtb_Sum1_idx_2;

  /* Sum: '<S21>/Sum1' incorporates:
   *  Constant: '<S21>/Constant2'
   */
  rtb_Gain = rtb_Divide2_f + 1.0;

  /* Gain: '<S21>/Gain1' */
  rtb_Divide2_f = rtb_Switch2_ejy_tmp;

  /* Saturate: '<S21>/Saturation3' */
  if (rtb_Sum_mf <= 1.0) {
    rtb_Sum_mf = 1.0;
  }

  /* End of Saturate: '<S21>/Saturation3' */

  /* Product: '<S21>/Divide2' incorporates:
   *  Constant: '<S21>/Constant'
   *  Product: '<S21>/Divide1'
   *  Sum: '<S21>/Sum2'
   */
  u0 = rtb_Gain * rtb_kW2W * Gen2_ref_B->T2s_filt.Switch *
    (Gen2_ref_B->Pel_filt.Switch + rtb_Divide2_f) * 12.566370614359172 * (1.0 /
    rtb_Sum_mf);

  /* Saturate: '<S21>/Saturation2' */
  if (u0 > 1.0) {
    /* DataTypeConversion: '<Root>/Data Type Conversion1' */
    Gen2_ref_B->DataTypeConversion1 = 1.0F;
  } else if (u0 < 0.0001) {
    /* DataTypeConversion: '<Root>/Data Type Conversion1' */
    Gen2_ref_B->DataTypeConversion1 = 0.0001F;
  } else {
    /* DataTypeConversion: '<Root>/Data Type Conversion1' */
    Gen2_ref_B->DataTypeConversion1 = (real32_T)u0;
  }

  /* End of Saturate: '<S21>/Saturation2' */
  /* End of Outputs for SubSystem: '<Root>/brake eff estimate' */

  /* S-Function (bur_out): '<Root>/Output' */
  inst->rEtaBrakeEst = Gen2_ref_B->DataTypeConversion1;

  /* DataTypeConversion: '<S22>/Data Type Conversion' incorporates:
   *  Constant: '<S47>/Constant'
   *  DiscreteIntegrator: '<S22>/Discrete-Time Integrator'
   *  RelationalOperator: '<S47>/Compare'
   */
  rtb_Sum_mf = (Gen2_ref_DWork->DiscreteTimeIntegrator_DSTATE_i > 0.0);

  /* Product: '<S22>/Product1' */
  rtb_Divide2_f = rtb_Gain_kp * Gen2_ref_B->BusInput3.bdcWgv.rKiWgvTcOvrspdCtrl;

  /* Product: '<S22>/Product2' */
  rtb_Gain = Gen2_ref_B->BusInput3.bdcWgv.rIntDischargeTcOvrspedCtrl *
    rtb_Sum_mf;

  /* Saturate: '<S22>/Saturation2' */
  if (rtb_Divide2_f <= 0.0) {
    delta_y = 0.0;
  } else {
    delta_y = rtb_Divide2_f;
  }

  /* End of Saturate: '<S22>/Saturation2' */

  /* DataTypeConversion: '<S48>/Data Type Conversion1' incorporates:
   *  Constant: '<S66>/Constant'
   *  DiscreteIntegrator: '<S48>/Discrete-Time Integrator'
   *  RelationalOperator: '<S66>/Compare'
   */
  rtb_Sum_mf = (Gen2_ref_DWork->DiscreteTimeIntegrator_DSTAT_ac > 0.0);

  /* Product: '<S48>/Product3' */
  rtb_Divide2_f = rtb_Divide3_k *
    Gen2_ref_B->BusInput3.bdcMisc.rKiSurgeProtectSL;

  /* Sum: '<S48>/Sum11' incorporates:
   *  Product: '<S48>/Product4'
   */
  rtb_Switch_eu = rtb_Divide2_f -
    Gen2_ref_B->BusInput3.bdcMisc.rIntDischargeSurgeCtrl * rtb_Sum_mf;

  /* Sum: '<S26>/Sum2' incorporates:
   *  MATLAB Function: '<S26>/fb_err'
   *  Product: '<S26>/Product1'
   */
  rtb_Switch1_mm = err * rtb_Pa2bar + FILT_IN;

  /* Saturate: '<S132>/Saturation' */
  if (Gen2_ref_B->BusInput3.bdcMisc.rTiF_Pr_p2s > 1000.0) {
    FILT_IN = 1000.0;
  } else if (Gen2_ref_B->BusInput3.bdcMisc.rTiF_Pr_p2s < 0.001) {
    FILT_IN = 0.001;
  } else {
    FILT_IN = Gen2_ref_B->BusInput3.bdcMisc.rTiF_Pr_p2s;
  }

  /* End of Saturate: '<S132>/Saturation' */

  /* Product: '<S132>/Divide' incorporates:
   *  DiscreteIntegrator: '<S132>/Discrete-Time Integrator'
   *  Sum: '<S132>/Sum4'
   */
  rtb_Gain1_fr = (Gen2_ref_B->p2s_filt.Switch -
                  Gen2_ref_DWork->DiscreteTimeIntegrator_DSTATE_g) / FILT_IN;

  /* Abs: '<S135>/Abs' incorporates:
   *  Abs: '<S742>/Abs'
   */
  FILT_IN = rtb_Switch_dz_tmp;

  /* Switch: '<S135>/Switch' incorporates:
   *  Constant: '<S135>/Constant2'
   *  RelationalOperator: '<S135>/Relational Operator'
   */
  if (2.2204460492503131E-16 >= FILT_IN) {
    rtb_bResetHlci_0 = 2.2204460492503131E-16;
  } else {
    rtb_bResetHlci_0 = Gen2_ref_B->BusInput3.eng.Ts;
  }

  /* End of Switch: '<S135>/Switch' */

  /* Product: '<S133>/Divide' incorporates:
   *  Logic: '<S133>/Logical Operator2'
   *  Logic: '<S133>/Logical Operator3'
   *  UnitDelay: '<S133>/Unit Delay'
   */
  rtb_Saturation = (real_T)((!rtb_LogicalOperator1_ix) &&
    Gen2_ref_DWork->UnitDelay_DSTATE_o) / rtb_bResetHlci_0;

  /* Switch: '<S161>/Switch' incorporates:
   *  Constant: '<S161>/Constant'
   */
  if (rtb_LogicalOperator3_k) {
    rtb_Sum8_m = rtb_Add2;
  } else {
    rtb_Sum8_m = 0.0;
  }

  /* End of Switch: '<S161>/Switch' */

  /* Product: '<S5>/Divide3' */
  rtb_Divide3_e[0] = Gen2_ref_B->BusInput.IN_EC_rGT_RatioMix_TC2 *
    rtb_Divide_ab[0];
  rtb_Divide3_e[1] = Gen2_ref_B->BusInput.IN_EC_rGT_RatioMix_TC2 *
    rtb_Divide_ab[1];
  rtb_Divide3_e[2] = Gen2_ref_B->BusInput.IN_EC_rGT_RatioMix_TC2 *
    rtb_Divide_ab[2];
  rtb_Divide3_e[3] = Gen2_ref_B->BusInput.IN_EC_rGT_RatioMix_TC2 *
    rtb_Divide_ab[3];

  /* Switch: '<S345>/Switch2' incorporates:
   *  Constant: '<S345>/Constant4'
   *  Product: '<S345>/Divide'
   *  Saturate: '<S345>/Saturation'
   */
  if (Gen2_ref_B->BusInput.bActive_p2sMan) {
    rtb_DataTypeConversion15 = -100.0;
  } else {
    if (Gen2_ref_B->BusInput3.traj.rTiLEANOXman <= 0.01) {
      /* Saturate: '<S345>/Saturation' */
      rtb_bResetHlci_0 = 0.01;
    } else {
      /* Saturate: '<S345>/Saturation' */
      rtb_bResetHlci_0 = Gen2_ref_B->BusInput3.traj.rTiLEANOXman;
    }

    rtb_DataTypeConversion15 = 1.0 / rtb_bResetHlci_0;
  }

  /* End of Switch: '<S345>/Switch2' */

  /* Outputs for Atomic SubSystem: '<S8>/BDC_Trajectory' */
  /* DiscreteIntegrator: '<S417>/Discrete-Time Integrator' */
  if (rtb_bResetHlci || (Gen2_ref_DWork->DiscreteTimeIntegrator_PrevR_ly != 0))
  {
    Gen2_ref_DWork->DiscreteTimeIntegrator_DSTATE_b = 1.0;
  }

  if (Gen2_ref_DWork->DiscreteTimeIntegrator_DSTATE_b >= 1.0) {
    Gen2_ref_DWork->DiscreteTimeIntegrator_DSTATE_b = 1.0;
  } else if (Gen2_ref_DWork->DiscreteTimeIntegrator_DSTATE_b <= 0.0) {
    Gen2_ref_DWork->DiscreteTimeIntegrator_DSTATE_b = 0.0;
  }

  /* Logic: '<S417>/Logical Operator' incorporates:
   *  Constant: '<S417>/Constant2'
   *  DiscreteIntegrator: '<S417>/Discrete-Time Integrator'
   *  RelationalOperator: '<S417>/Relational Operator'
   */
  rtb_LogicalOperator5_mv = ((0.99 <=
    Gen2_ref_DWork->DiscreteTimeIntegrator_DSTATE_b) || rtb_bResetHlci);

  /* Product: '<S434>/delta rise limit' */
  FILT_IN = rtb_Divide_mr_tmp_0;

  /* Delay: '<S434>/Delay' */
  Gen2_ref_DWork->icLoad_mu = ((((Gen2_ref_PrevZCSigState->Delay_Reset_ZCE_mt ==
    1) != (int32_T)rtb_LogicalOperator5_mv) &&
    (Gen2_ref_PrevZCSigState->Delay_Reset_ZCE_mt != 3)) ||
    rtb_LogicalOperator5_mv || Gen2_ref_DWork->icLoad_mu);
  Gen2_ref_PrevZCSigState->Delay_Reset_ZCE_mt = rtb_LogicalOperator5_mv;
  if (Gen2_ref_DWork->icLoad_mu) {
    Gen2_ref_DWork->Delay_DSTATE_h4 = rtb_bar2Pa6;
  }

  /* Sum: '<S434>/Difference Inputs1' incorporates:
   *  Delay: '<S434>/Delay'
   *  Switch: '<S434>/etaVolConst'
   */
  rtb_bar2Pa6 -= Gen2_ref_DWork->Delay_DSTATE_h4;

  /* Switch: '<S437>/Switch2' incorporates:
   *  RelationalOperator: '<S437>/LowerRelop1'
   */
  if (!(rtb_bar2Pa6 > FILT_IN)) {
    /* Product: '<S434>/delta fall limit' incorporates:
     *  Gain: '<S417>/Gain15'
     *  SampleTimeMath: '<S434>/sample time'
     *
     * About '<S434>/sample time':
     *  y = K where K = ( w * Ts )
     */
    rtb_Gain2_ao = -rtb_Switch_ct_tmp * 0.01;

    /* Switch: '<S437>/Switch' incorporates:
     *  RelationalOperator: '<S437>/UpperRelop'
     */
    if (rtb_bar2Pa6 < rtb_Gain2_ao) {
      FILT_IN = rtb_Gain2_ao;
    } else {
      FILT_IN = rtb_bar2Pa6;
    }

    /* End of Switch: '<S437>/Switch' */
  }

  /* End of Switch: '<S437>/Switch2' */

  /* Sum: '<S434>/Difference Inputs2' incorporates:
   *  Delay: '<S434>/Delay'
   */
  rtb_bar2Pa6 = FILT_IN + Gen2_ref_DWork->Delay_DSTATE_h4;

  /* Outputs for Atomic SubSystem: '<S417>/p2sfilt' */
  Gen2_ref_N_TC_HP_filt(rtb_bar2Pa6, Gen2_ref_B->BusInput3.traj.rTiF_Pr_p2s_Man,
                        rtb_LogicalOperator5_mv, &Gen2_ref_B->p2sfilt_b,
                        &Gen2_ref_DWork->p2sfilt_b, inst);

  /* End of Outputs for SubSystem: '<S417>/p2sfilt' */

  /* Sum: '<S417>/Sum1' incorporates:
   *  Constant: '<S417>/Constant1'
   *  DiscreteIntegrator: '<S417>/Discrete-Time Integrator'
   *  Product: '<S417>/Product'
   *  Product: '<S417>/Product1'
   *  Sum: '<S417>/Sum'
   */
  rtb_Divide2_f = (1.0 - Gen2_ref_DWork->DiscreteTimeIntegrator_DSTATE_b) *
    Gen2_ref_B->p2sfilt_b.Switch +
    Gen2_ref_DWork->DiscreteTimeIntegrator_DSTATE_b * rtb_mbar2pa_i;

  /* Switch: '<S417>/Switch2' incorporates:
   *  Constant: '<S417>/Constant4'
   *  Product: '<S417>/Divide'
   *  Saturate: '<S417>/Saturation'
   */
  if (Gen2_ref_B->BusInput.bActive_p2sMan) {
    rtb_Gain2_ao = -100.0;
  } else {
    if (Gen2_ref_B->BusInput3.traj.rTiLEANOXman <= 0.01) {
      /* Saturate: '<S417>/Saturation' */
      rtb_bResetHlci_0 = 0.01;
    } else {
      /* Saturate: '<S417>/Saturation' */
      rtb_bResetHlci_0 = Gen2_ref_B->BusInput3.traj.rTiLEANOXman;
    }

    rtb_Gain2_ao = 1.0 / rtb_bResetHlci_0;
  }

  /* End of Switch: '<S417>/Switch2' */

  /* Update for DiscreteIntegrator: '<S417>/Discrete-Time Integrator' incorporates:
   *  Logic: '<S743>/Logical Operator'
   */
  Gen2_ref_DWork->DiscreteTimeIntegrator_DSTATE_b += 0.01 * rtb_Gain2_ao;
  if (Gen2_ref_DWork->DiscreteTimeIntegrator_DSTATE_b >= 1.0) {
    Gen2_ref_DWork->DiscreteTimeIntegrator_DSTATE_b = 1.0;
  } else if (Gen2_ref_DWork->DiscreteTimeIntegrator_DSTATE_b <= 0.0) {
    Gen2_ref_DWork->DiscreteTimeIntegrator_DSTATE_b = 0.0;
  }

  /* Outputs for Atomic SubSystem: '<S737>/Filter' */
  Gen2_ref_DWork->DiscreteTimeIntegrator_PrevR_ly = (int8_T)rtb_bResetHlci;

  /* End of Update for DiscreteIntegrator: '<S417>/Discrete-Time Integrator' */
  /* End of Outputs for SubSystem: '<S737>/Filter' */

  /* Update for Delay: '<S434>/Delay' */
  Gen2_ref_DWork->icLoad_mu = false;
  Gen2_ref_DWork->Delay_DSTATE_h4 = rtb_bar2Pa6;

  /* End of Outputs for SubSystem: '<S8>/BDC_Trajectory' */

  /* Sum: '<S427>/Sum5' incorporates:
   *  Constant: '<S427>/Constant6'
   */
  FILT_IN = Gen2_ref_B->BusInput3.LR.rTiAvoidTrigMisf + 0.01;

  /* DataTypeConversion: '<S427>/Data Type Conversion5' */
  rtb_rPos_CBV3 = (real32_T)FILT_IN;

  /* Sum: '<S427>/Sum7' incorporates:
   *  Constant: '<S427>/Constant6'
   *  Sum: '<S427>/Sum5'
   */
  FILT_IN = Gen2_ref_B->BusInput3.LR.rTiAvoidTrigMisf + 0.01;

  /* DataTypeConversion: '<S427>/Data Type Conversion6' */
  rtb_TOF2_PT = (real32_T)FILT_IN;

  /* Gain: '<S427>/Gain' */
  FILT_IN = 0.001 * rtb_Switch_i5[3];

  /* Abs: '<S507>/Abs' */
  rtb_Sum_mf = rtb_Product1_e_tmp;

  /* Switch: '<S507>/Switch' incorporates:
   *  Constant: '<S507>/Constant2'
   *  RelationalOperator: '<S507>/Relational Operator'
   */
  if (2.2204460492503131E-16 >= rtb_Sum_mf) {
    rtb_bResetHlci_0 = 2.2204460492503131E-16;
  } else {
    rtb_bResetHlci_0 = Gen2_ref_B->BusInput3.eng.rP_Nom;
  }

  /* End of Switch: '<S507>/Switch' */

  /* Product: '<S427>/Divide1' */
  rtb_bar2Pa6 = FILT_IN / rtb_bResetHlci_0;

  /* Outputs for Atomic SubSystem: '<S427>/TOF' */
  Gen2_ref_TOF_c(rtb_TOF_IN, rtb_rPos_CBV3, &Gen2_ref_B->TOF_c,
                 &Gen2_ref_DWork->TOF_c, inst);

  /* End of Outputs for SubSystem: '<S427>/TOF' */

  /* Outputs for Atomic SubSystem: '<S427>/TOF2' */
  Gen2_ref_TOF_c(Gen2_ref_B->TP_Misfire_ON.LogicalOperator1, rtb_TOF2_PT,
                 &Gen2_ref_B->TOF2_d, &Gen2_ref_DWork->TOF2_d, inst);

  /* End of Outputs for SubSystem: '<S427>/TOF2' */

  /* Abs: '<S583>/Abs' */
  FILT_IN = fabs(Gen2_ref_B->BusInput3.SkipF.rTiF_Lam);

  /* Switch: '<S583>/Switch' incorporates:
   *  Constant: '<S583>/Constant2'
   *  RelationalOperator: '<S583>/Relational Operator'
   */
  if (2.2204460492503131E-16 >= FILT_IN) {
    rtb_bResetHlci_0 = 2.2204460492503131E-16;
  } else {
    rtb_bResetHlci_0 = Gen2_ref_B->BusInput3.SkipF.rTiF_Lam;
  }

  /* End of Switch: '<S583>/Switch' */

  /* Product: '<S579>/Divide' incorporates:
   *  DiscreteIntegrator: '<S579>/Discrete-Time Integrator'
   *  Sum: '<S579>/Sum4'
   */
  rtb_Gain2_ao = (rtb_Sum2_kg - Gen2_ref_DWork->DiscreteTimeIntegrator_DSTATE_m)
    / rtb_bResetHlci_0;

  /* Product: '<S586>/Product3' */
  rtb_p2s = Gen2_ref_B->BusInput3.SkipF.rKiTrackLam * rtb_W2kW_o;

  /* DataTypeConversion: '<S581>/Data Type Conversion13' */
  FILT_IN = Gen2_ref_B->BusInput3.SkipF.iNr_cycles_ignOFF;

  /* Bias: '<S608>/Bias' incorporates:
   *  Gain: '<S581>/ to Hz'
   *  Gain: '<S581>/Hz to cycle period2'
   *  Product: '<S581>/Divide7'
   */
  FILT_IN = FILT_IN / rtb_Saturation_o * 60.0 * 2.0 + -0.01;

  /* Abs: '<S612>/Abs' */
  rtb_Sum_mf = fabs(FILT_IN);

  /* RelationalOperator: '<S612>/Relational Operator' incorporates:
   *  Constant: '<S612>/Constant2'
   */
  rtb_TOF_IN = (2.2204460492503131E-16 >= rtb_Sum_mf);

  /* Sum: '<S608>/Sum1' */
  rtb_Sum_mf = Gen2_ref_B->BusInput3.SkipF.rThrsh_PulseGenerator_reset -
    Gen2_ref_B->BusInput3.SkipF.rThrsh_PulseGenerator_trigger;

  /* Switch: '<S612>/Switch' incorporates:
   *  Constant: '<S612>/Constant2'
   */
  if (rtb_TOF_IN) {
    FILT_IN = 2.2204460492503131E-16;
  }

  /* End of Switch: '<S612>/Switch' */

  /* Product: '<S608>/Product1' */
  rtb_Switch2_g3 = rtb_Sum_mf / FILT_IN;

  /* RelationalOperator: '<S608>/Relational Operator1' incorporates:
   *  DiscreteIntegrator: '<S608>/Discrete-Time Integrator'
   */
  rtb_TOF_IN = (Gen2_ref_DWork->DiscreteTimeIntegrator_DSTAT_h5 >=
                Gen2_ref_B->BusInput3.SkipF.rThrsh_PulseGenerator_reset);

  /* Outputs for Atomic SubSystem: '<S633>/Filter' */
  Gen2_ref_Filter3(Gen2_ref_B->sf_MATLABFunction_kd.y,
                   Gen2_ref_B->BusInput3.SkipF.rTiF_stat,
                   Gen2_ref_ConstB.Constant3, rtb_bResetHlci,
                   &Gen2_ref_B->Filter_pj, &Gen2_ref_DWork->Filter_pj, inst);

  /* End of Outputs for SubSystem: '<S633>/Filter' */

  /* MATLAB Function: '<S431>/ref traj' */
  if ((!Gen2_ref_DWork->x_not_empty_i) || rtb_bResetHlci) {
    Gen2_ref_DWork->x_d = rtb_Gain3;
    Gen2_ref_DWork->x_not_empty_i = true;
  }

  if ((Gen2_ref_B->BusInput3.traj.rTi_BDC >= Ts_tmp) ||
      rtb_LogicalOperator5_g_tmp) {
    rtb_bResetHlci_0 = Gen2_ref_B->BusInput3.traj.rTi_BDC;
  } else {
    rtb_bResetHlci_0 = Ts_tmp;
  }

  rtb_Switch2_a = rtb_Product_m[0] - Gen2_ref_DWork->x_d;
  u0 = 1.0 / rtb_bResetHlci_0 * rtb_Switch2_a;
  if ((Gen2_ref_B->BusInput3.traj.rTi_BDC >= Ts_tmp) ||
      rtb_LogicalOperator5_g_tmp) {
    rtb_bResetHlci_0 = Gen2_ref_B->BusInput3.traj.rTi_BDC;
  } else {
    rtb_bResetHlci_0 = Ts_tmp;
  }

  FILT_IN = 1.0 / rtb_bResetHlci_0 * rtb_Switch2_a;
  if ((u0 >= FILT_IN) || rtIsNaN(FILT_IN)) {
    FILT_IN = u0;
  }

  if (FILT_IN > 0.0) {
    u0 = FILT_IN * Ts_tmp + Gen2_ref_DWork->x_d;
    rtb_Divide2_a = rtb_Gain3 + Gen2_ref_B->BusInput3.traj.rPrR_delta_p2s;
    if ((u0 <= rtb_Divide2_a) || rtIsNaN(rtb_Divide2_a)) {
      rtb_Divide2_a = u0;
    }
  } else {
    u0 = FILT_IN * Ts_tmp + Gen2_ref_DWork->x_d;
    rtb_Divide2_a = rtb_Gain3 - Gen2_ref_B->BusInput3.traj.rPrR_delta_p2s;
    if ((u0 >= rtb_Divide2_a) || rtIsNaN(rtb_Divide2_a)) {
      rtb_Divide2_a = u0;
    }
  }

  Gen2_ref_DWork->x_d = rtb_Divide2_a;

  /* SignalConversion generated from: '<S431>/Delay' */
  rtb_Divide_ab[0] = rtb_Divide2_a;
  rtb_Divide_ab[1] = Gen2_ref_B->Filter_bd.Switch;
  rtb_Divide_ab[3] = Gen2_ref_B->sf_MATLABFunction_kd.y;

  /* Sum: '<S634>/Sum1' */
  FILT_IN = rtb_Product1_c1_tmp;

  /* Outputs for Atomic SubSystem: '<S634>/TON' */
  Gen2_ref_TON_1(rtb_bTriger_IT_LJ, Gen2_ref_B->BusInput3.ITC.rITCtransTON,
                 &Gen2_ref_B->TON_c, &Gen2_ref_DWork->TON_c, inst);

  /* End of Outputs for SubSystem: '<S634>/TON' */

  /* Switch: '<S634>/Switch2' incorporates:
   *  Abs: '<S634>/Abs'
   *  Logic: '<S634>/Logical Operator1'
   *  Logic: '<S634>/Logical Operator5'
   *  RelationalOperator: '<S634>/Relational Operator3'
   */
  rtb_LogicalOperator5_mv = ((!rtb_bResetHlci) &&
    ((!Gen2_ref_B->TON_c.LogicalOperator3) ||
     (!(Gen2_ref_B->BusInput3.ITC.rITCtransNthrsh > fabs(FILT_IN)))) &&
    rtb_bTriger_IT_LJ);

  /* Switch: '<S714>/Switch6' incorporates:
   *  Constant: '<S714>/Constant'
   *  Constant: '<S715>/Constant'
   *  Logic: '<S714>/Logical Operator4'
   *  Switch: '<S715>/Switch6'
   */
  if (!rtb_LogicalOperator2_ov) {
    /* Switch: '<S714>/Switch1' incorporates:
     *  DiscreteIntegrator: '<S714>/Discrete-Time Integrator'
     *  Gain: '<S714>/Gain2'
     */
    if (rtb_Switch2_au) {
      /* Switch: '<S636>/Switch8' incorporates:
       *  Gain: '<S636>/Gain3'
       *  Logic: '<S636>/Logical Operator7'
       */
      if (Gen2_ref_B->BusInput3.SpeedCtrl.bKF_KeLearn_boost &&
          Gen2_ref_B->BusInput3.SpeedCtrl.bKF_act) {
        rtb_bResetHlci_0 = -rtb_Switch1_cl[0];
      } else {
        rtb_bResetHlci_0 = rtb_Switch_dhr;
      }

      /* End of Switch: '<S636>/Switch8' */

      /* Product: '<S714>/Product' incorporates:
       *  Abs: '<S714>/Abs'
       *  Gain: '<S714>/Gain1'
       */
      rtb_Switch_ks = -fabs(Gen2_ref_B->BusInput3.SpeedCtrl.rKeAdaptGain) *
        rtb_bResetHlci_0;

      /* Switch: '<S721>/Switch2' incorporates:
       *  Gain: '<S714>/Gain'
       *  RelationalOperator: '<S721>/LowerRelop1'
       *  RelationalOperator: '<S721>/UpperRelop'
       *  Switch: '<S721>/Switch'
       */
      if (rtb_Switch_ks > Gen2_ref_B->BusInput3.SpeedCtrl.rKeAdaptRL) {
        rtb_Switch_ks = Gen2_ref_B->BusInput3.SpeedCtrl.rKeAdaptRL;
      } else if (rtb_Switch_ks < -Gen2_ref_B->BusInput3.SpeedCtrl.rKeAdaptRL) {
        /* Switch: '<S721>/Switch' incorporates:
         *  Gain: '<S714>/Gain'
         */
        rtb_Switch_ks = -Gen2_ref_B->BusInput3.SpeedCtrl.rKeAdaptRL;
      }

      /* End of Switch: '<S721>/Switch2' */
    } else {
      rtb_Switch_ks = -Gen2_ref_DWork->DiscreteTimeIntegrator_DSTATE_l;
    }

    /* End of Switch: '<S714>/Switch1' */

    /* Switch: '<S715>/Switch1' incorporates:
     *  DiscreteIntegrator: '<S715>/Discrete-Time Integrator'
     *  Gain: '<S715>/Gain2'
     */
    if (rtb_Switch3_le) {
      /* Switch: '<S636>/Switch9' incorporates:
       *  Gain: '<S636>/Gain4'
       *  Logic: '<S636>/Logical Operator8'
       */
      if (Gen2_ref_B->BusInput3.SpeedCtrl.bKF_KeLearn_power &&
          Gen2_ref_B->BusInput3.SpeedCtrl.bKF_act) {
        rtb_Switch_dhr = -rtb_Switch1_cl[0];
      }

      /* End of Switch: '<S636>/Switch9' */

      /* Product: '<S715>/Product' incorporates:
       *  Abs: '<S715>/Abs'
       *  Gain: '<S715>/Gain1'
       */
      rtb_Divide2_a = -fabs(Gen2_ref_B->BusInput3.SpeedCtrl.rKeAdaptGain) *
        rtb_Switch_dhr;

      /* Switch: '<S725>/Switch2' incorporates:
       *  Gain: '<S715>/Gain'
       *  RelationalOperator: '<S725>/LowerRelop1'
       *  RelationalOperator: '<S725>/UpperRelop'
       *  Switch: '<S725>/Switch'
       */
      if (rtb_Divide2_a > Gen2_ref_B->BusInput3.SpeedCtrl.rKeAdaptRL) {
        rtb_Divide2_a = Gen2_ref_B->BusInput3.SpeedCtrl.rKeAdaptRL;
      } else if (rtb_Divide2_a < -Gen2_ref_B->BusInput3.SpeedCtrl.rKeAdaptRL) {
        /* Switch: '<S725>/Switch' incorporates:
         *  Gain: '<S715>/Gain'
         */
        rtb_Divide2_a = -Gen2_ref_B->BusInput3.SpeedCtrl.rKeAdaptRL;
      }

      /* End of Switch: '<S725>/Switch2' */
    } else {
      rtb_Divide2_a = -Gen2_ref_DWork->DiscreteTimeIntegrator_DSTATE_e;
    }

    /* End of Switch: '<S715>/Switch1' */
  } else {
    rtb_Switch_ks = 0.0;
    rtb_Divide2_a = 0.0;
  }

  /* End of Switch: '<S714>/Switch6' */

  /* Switch: '<S747>/Switch1' incorporates:
   *  Constant: '<S747>/Constant'
   *  Logic: '<S747>/Logical Operator'
   *  Logic: '<S747>/Logical Operator1'
   *  Switch: '<S747>/Switch2'
   *  UnitDelay: '<S641>/Unit Delay2'
   */
  if (!Gen2_ref_DWork->UnitDelay2_DSTATE_d2) {
    /* Switch: '<S747>/Switch3' */
    if (Gen2_ref_B->BusInput3.SpeedCtrl.bGS_Kspeed_iLQR) {
      /* S-Function (sfix_look1_dyn): '<S747>/gain scheduling Kspeed' */
      /* Dynamic Look-Up Table Block: '<S747>/gain scheduling Kspeed'
       * Input0  Data Type:  Floating Point real_T
       * Input1  Data Type:  Floating Point real_T
       * Input2  Data Type:  Floating Point real_T
       * Output0 Data Type:  Floating Point real_T
       * Lookup Method: Linear_Endpoint
       *
       */
      LookUp_real_T_real_T( &(rtb_gainschedulingKspeed),
                           &Gen2_ref_B->BusInput3.SpeedCtrl.refPoint_iLQR_Kspeed_y
                           [0], rtb_Gain3,
                           &Gen2_ref_B->BusInput3.SpeedCtrl.refPoint_iLQR_Kspeed_x
                           [0], 6U, inst);
      FILT_IN = rtb_gainschedulingKspeed;
    } else {
      FILT_IN = Gen2_ref_B->BusInput3.SpeedCtrl.rGain_ss_speed_iLQR;
    }

    /* End of Switch: '<S747>/Switch3' */
  } else if (Gen2_ref_DWork->UnitDelay2_DSTATE_d2 &&
             Gen2_ref_B->TON_d.LogicalOperator3) {
    /* Switch: '<S747>/Switch2' */
    FILT_IN = Gen2_ref_B->BusInput3.SpeedCtrl.rGain_ss_speed_iLQR_back;
  } else {
    FILT_IN = 0.0;
  }

  /* End of Switch: '<S747>/Switch1' */

  /* Switch: '<S747>/Switch4' incorporates:
   *  Constant: '<S747>/Constant'
   */
  if (rtb_LogicalOperator3_b) {
    rtb_Sum_mf = 0.0;
  } else {
    rtb_Sum_mf = Gen2_ref_B->BusInput3.SpeedCtrl.rGain_ss_boost_iLQR;
  }

  /* End of Switch: '<S747>/Switch4' */

  /* Switch: '<S641>/Switch' incorporates:
   *  Gain: '<S8>/pa2bar   '
   */
  if (Gen2_ref_B->BusInput3.SpeedCtrl.bSepEmisCtrl) {
    rtb_Abs = 1.0E-5 * rtb_Divide2_f;
  }

  /* End of Switch: '<S641>/Switch' */

  /* Sum: '<S748>/Sum3' incorporates:
   *  DiscreteIntegrator: '<S748>/Discrete-Time Integrator4'
   */
  rtb_MinMax_n = (Gen2_ref_DWork->DiscreteTimeIntegrator4_DSTATE + rtb_Abs) -
    rtb_Gain3;

  /* Switch: '<S752>/Switch2' */
  if (Gen2_ref_B->BusInput3.SpeedCtrl.bAW_iLQR_LEANOX) {
    /* RelationalOperator: '<S752>/Relational Operator1' incorporates:
     *  Constant: '<S752>/Constant4'
     *  Product: '<S752>/Divide1'
     *  Sum: '<S752>/Sum'
     */
    rtb_LogicalOperator2_fy = (rtb_Divide3_ep / rtb_PrefOut >= 1.0 - rtb_PactOut);

    /* Switch: '<S752>/Switch' incorporates:
     *  Constant: '<S752>/Constant'
     *  Constant: '<S752>/Constant1'
     *  Logic: '<S752>/Logical Operator'
     *  RelationalOperator: '<S752>/Relational Operator'
     *  UnitDelay: '<Root>/Unit Delay3'
     */
    if ((Gen2_ref_DWork->UnitDelay3_DSTATE <= rtb_Switch2_ejy_tmp_0) &&
        rtb_LogicalOperator2_fy) {
      rtb_Divide2_f = 0.0;
    } else {
      rtb_Divide2_f = 1.0E+6;
    }

    /* End of Switch: '<S752>/Switch' */

    /* Switch: '<S755>/Switch2' incorporates:
     *  RelationalOperator: '<S755>/LowerRelop1'
     */
    if (!(rtb_MinMax_n > rtb_Divide2_f)) {
      /* Saturate: '<S752>/Saturation1' */
      if (Gen2_ref_B->BusInput3.bdcCbv.rPos_max > 1.0) {
        rtb_bResetHlci_0 = 1.0;
      } else if (Gen2_ref_B->BusInput3.bdcCbv.rPos_max < 0.1) {
        rtb_bResetHlci_0 = 0.1;
      } else {
        rtb_bResetHlci_0 = Gen2_ref_B->BusInput3.bdcCbv.rPos_max;
      }

      /* End of Saturate: '<S752>/Saturation1' */

      /* Switch: '<S752>/Switch1' incorporates:
       *  Constant: '<S752>/Constant2'
       *  Constant: '<S752>/Constant3'
       *  Constant: '<S752>/Constant4'
       *  Logic: '<S752>/Logical Operator1'
       *  Logic: '<S752>/Logical Operator2'
       *  Product: '<S752>/Divide'
       *  RelationalOperator: '<S752>/Relational Operator2'
       *  RelationalOperator: '<S752>/Relational Operator3'
       *  Sum: '<S752>/Sum'
       *  UnitDelay: '<Root>/Unit Delay3'
       */
      if ((Gen2_ref_DWork->UnitDelay3_DSTATE / rtb_bResetHlci_0 >= 1.0 -
           rtb_PactOut) && ((rtb_Divide3_ep <= rtb_LogicalOperator1_js_tmp) ||
                            rtb_LogicalOperator2_fy)) {
        rtb_Divide2_f = 0.0;
      } else {
        rtb_Divide2_f = -1.0E+6;
      }

      /* End of Switch: '<S752>/Switch1' */

      /* Switch: '<S755>/Switch' incorporates:
       *  RelationalOperator: '<S755>/UpperRelop'
       */
      if (!(rtb_MinMax_n < rtb_Divide2_f)) {
        rtb_Divide2_f = rtb_MinMax_n;
      }

      /* End of Switch: '<S755>/Switch' */
    }
  } else {
    rtb_Divide2_f = rtb_MinMax_n;
  }

  /* Switch: '<S756>/Switch2' incorporates:
   *  RelationalOperator: '<S756>/LowerRelop1'
   *  RelationalOperator: '<S756>/UpperRelop'
   *  Switch: '<S756>/Switch'
   */
  if (Gen2_ref_B->Filter_bd.Switch > rtb_Switch2_n5) {
    rtb_Sum2_a1 = rtb_Switch2_n5;
  } else if (Gen2_ref_B->Filter_bd.Switch < rtb_Switch1_k) {
    /* Switch: '<S756>/Switch' */
    rtb_Sum2_a1 = rtb_Switch1_k;
  } else {
    rtb_Sum2_a1 = Gen2_ref_B->Filter_bd.Switch;
  }

  /* End of Switch: '<S756>/Switch2' */

  /* Sum: '<S753>/Sum2' incorporates:
   *  Product: '<S753>/Product'
   *  Sum: '<S753>/Sum1'
   */
  rtb_Sum2_a1 = (rtb_Sum2_a1 - Gen2_ref_B->Filter_bd.Switch) *
    Gen2_ref_B->BusInput3.SpeedCtrl.rGain_LEANOX_AW_iLQR + rtb_MinMax_n;

  /* Switch: '<S748>/Switch3' incorporates:
   *  Constant: '<S748>/Constant5'
   *  Logic: '<S748>/Logical Operator7'
   *  Sum: '<S748>/Sum'
   */
  if (Gen2_ref_B->BusInput3.SpeedCtrl.bAWLam_iLQR && (rtb_kW2W1_h != 0.0)) {
    rtb_Product4_d = 0.0;
  } else {
    rtb_Product4_d = rtb_Saturation6_tmp;
  }

  /* End of Switch: '<S748>/Switch3' */

  /* Switch: '<S754>/Switch2' incorporates:
   *  RelationalOperator: '<S754>/LowerRelop1'
   *  Sum: '<S748>/Sum'
   */
  if (!(rtb_Saturation6_tmp > rtb_Product4_d)) {
    /* Switch: '<S748>/Switch4' incorporates:
     *  Constant: '<S748>/Constant5'
     *  Logic: '<S748>/Logical Operator8'
     */
    if ((rtb_Gain6_b != 0.0) &&
        Gen2_ref_B->BusInput3.SpeedCtrl.bAWLam_iLQR_uplim) {
      rtb_MinMax_n = 0.0;
    } else {
      rtb_MinMax_n = rtb_Saturation6_tmp;
    }

    /* End of Switch: '<S748>/Switch4' */

    /* Switch: '<S754>/Switch' incorporates:
     *  RelationalOperator: '<S754>/UpperRelop'
     */
    if (rtb_Saturation6_tmp < rtb_MinMax_n) {
      rtb_Product4_d = rtb_MinMax_n;
    } else {
      rtb_Product4_d = rtb_Saturation6_tmp;
    }

    /* End of Switch: '<S754>/Switch' */
  }

  /* End of Switch: '<S754>/Switch2' */

  /* Product: '<S748>/Product' */
  rtb_MinMax_n = rtb_Product4_d * FILT_IN;

  /* Product: '<S748>/Product1' */
  rtb_Divide2_f *= rtb_Sum_mf;

  /* Product: '<S748>/Product2' incorporates:
   *  Sum: '<S748>/Sum1'
   */
  rtb_Pa2bar_k = (rtb_Gain2_cm - Gen2_ref_B->Filter_pj.Switch) *
    Gen2_ref_B->BusInput3.SpeedCtrl.rGain_ss_Nskip_iLQR;

  /* Product: '<S748>/Product3' */
  rtb_Product1 = Gen2_ref_B->BusInput3.SpeedCtrl.rGain_ss_LEANOX_iLQR *
    rtb_Sum2_a1;

  /* Product: '<S748>/Product4' */
  rtb_Product4_d *= Gen2_ref_B->BusInput3.SpeedCtrl.rGain_ss_speed2boost_iLQR;

  /* Switch: '<S748>/Switch5' incorporates:
   *  Gain: '<S748>/Gain2'
   *  Gain: '<S748>/Gain3'
   */
  if (rtb_Gain6_b != 0.0) {
    rtb_Divide3_d = -Gen2_ref_B->BusInput3.SpeedCtrl.rGainLamUplim2boost;
  } else {
    rtb_Divide3_d = 0.1 * Gen2_ref_B->BusInput3.SpeedCtrl.rGainLamUplim2boost;
  }

  /* End of Switch: '<S748>/Switch5' */

  /* Switch: '<S760>/Switch2' incorporates:
   *  Constant: '<S760>/Constant4'
   *  Product: '<S760>/Divide'
   *  Saturate: '<S760>/Saturation'
   */
  if (Gen2_ref_B->BusInput.bActive_p2sMan) {
    rtb_Divide_kp = -100.0;
  } else {
    if (Gen2_ref_B->BusInput3.traj.rTiLEANOXman <= 0.01) {
      /* Saturate: '<S760>/Saturation' */
      rtb_bResetHlci_0 = 0.01;
    } else {
      /* Saturate: '<S760>/Saturation' */
      rtb_bResetHlci_0 = Gen2_ref_B->BusInput3.traj.rTiLEANOXman;
    }

    rtb_Divide_kp = 1.0 / rtb_bResetHlci_0;
  }

  /* End of Switch: '<S760>/Switch2' */

  /* Switch: '<S761>/Switch1' incorporates:
   *  Constant: '<S761>/Constant'
   *  Logic: '<S761>/Logical Operator'
   *  Sum: '<S761>/Sum'
   */
  if (Gen2_ref_B->BusInput3.LoadEst.bCorrUnom &&
      Gen2_ref_B->TON2.LogicalOperator3) {
    rtb_rKK2_k = 1.0 - rtb_rKK2_k;
  } else {
    rtb_rKK2_k = Gen2_ref_B->Filter1_p.Switch;
  }

  /* End of Switch: '<S761>/Switch1' */

  /* Logic: '<S12>/Logical Operator' */
  rtb_LogicalOperator2_fy = !Gen2_ref_B->TON2.LogicalOperator3;

  /* Switch: '<S15>/Switch5' incorporates:
   *  UnitDelay: '<S15>/Unit Delay'
   */
  if (Gen2_ref_B->TON2.LogicalOperator3) {
    rtb_mbar2pa_g = r;
  } else {
    rtb_mbar2pa_g = Gen2_ref_DWork->UnitDelay_DSTATE_fm;
  }

  /* End of Switch: '<S15>/Switch5' */

  /* Switch: '<S15>/Switch4' incorporates:
   *  Constant: '<S15>/Pel_a (kW)1'
   *  Constant: '<S15>/Pel_a (kW)4'
   *  Logic: '<S15>/Logical Operator'
   *  RelationalOperator: '<S15>/Relational Operator'
   */
  if (Gen2_ref_B->BusInput3.leanox.bWGKorr &&
      (Gen2_ref_B->BusInput3.eng.rNum_WGV > 0.0)) {
    rtb_bResetHlci_0 = rtb_mbar2pa_g;
  } else {
    rtb_bResetHlci_0 = 0.0;
  }

  /* End of Switch: '<S15>/Switch4' */

  /* Outputs for Atomic SubSystem: '<S15>/Filter1' */
  Gen2_ref_N_TC_HP_filt(rtb_bResetHlci_0, Gen2_ref_B->BusInput3.leanox.rTiF_WG,
                        rtb_bResetBdc, &Gen2_ref_B->Filter1_fj,
                        &Gen2_ref_DWork->Filter1_fj, inst);

  /* End of Outputs for SubSystem: '<S15>/Filter1' */

  /* Saturate: '<S18>/Saturation1' */
  FILT_IN = rtb_deltafalllimit_ca;

  /* Saturate: '<S18>/Saturation2' */
  r = rtb_PrefOut;

  /* Product: '<S18>/Divide1' */
  rtb_PrefOut = Gen2_ref_B->sf_IntegerZOH.y / r;

  /* Saturate: '<S18>/Saturation' */
  r = rtb_PactOut;

  /* Sum: '<S18>/Sum1' */
  rtb_Sum_mf = Gen2_ref_B->BusInput3.bdcCbv.rPos_min + r;

  /* RelationalOperator: '<S18>/Relational Operator' */
  rtb_bCBV_min = (rtb_TmpSignalConversionAtSFun_p[0] <= rtb_Sum_mf);

  /* Sum: '<S18>/Sum2' */
  rtb_Sum_mf = Gen2_ref_B->BusInput3.bdcTv.rPos_min + r;

  /* Sum: '<S18>/Sum' incorporates:
   *  Constant: '<S18>/Constant4'
   */
  r = 1.0 - r;

  /* Logic: '<S18>/Logical Operator2' incorporates:
   *  RelationalOperator: '<S18>/Relational Operator1'
   *  RelationalOperator: '<S18>/Relational Operator3'
   */
  rtb_bTV_sat = ((Gen2_ref_B->sf_IntegerZOH.y <= rtb_Sum_mf) || (rtb_PrefOut >=
    r));

  /* UnitDelay: '<S10>/Unit Delay' */
  Gen2_ref_B->UnitDelay = Gen2_ref_DWork->UnitDelay_DSTATE_j;

  /* S-Function (bur_out): '<Root>/Output1' */
  inst->Version = Gen2_ref_B->UnitDelay;

  /* Update for UnitDelay: '<S427>/Unit Delay4' */
  Gen2_ref_DWork->TOF_state = Gen2_ref_B->TOF_c.LogicalOperator1;

  /* Update for Delay: '<S427>/Delay' */
  for (k = 0; k < 29; k++) {
    Gen2_ref_DWork->Delay_DSTATE[k] = Gen2_ref_DWork->Delay_DSTATE[k + 1];
  }

  Gen2_ref_DWork->Delay_DSTATE[29] = rtb_bar2Pa6;

  /* End of Update for Delay: '<S427>/Delay' */

  /* Update for Delay: '<S425>/Delay' */
  Gen2_ref_DWork->icLoad = false;
  for (i = 0; i < 6; i++) {
    Gen2_ref_DWork->Delay_DSTATE_o[i] = rtb_TmpSignalConversionAtDelayI[i];
  }

  /* End of Update for Delay: '<S425>/Delay' */

  /* Update for DiscreteIntegrator: '<S345>/Discrete-Time Integrator' incorporates:
   *  DiscreteIntegrator: '<S389>/Discrete-Time Integrator1'
   */
  Gen2_ref_DWork->DiscreteTimeIntegrator_DSTATE += 0.01 *
    rtb_DataTypeConversion15;
  if (Gen2_ref_DWork->DiscreteTimeIntegrator_DSTATE >= 1.0) {
    Gen2_ref_DWork->DiscreteTimeIntegrator_DSTATE = 1.0;
  } else if (Gen2_ref_DWork->DiscreteTimeIntegrator_DSTATE <= 0.0) {
    Gen2_ref_DWork->DiscreteTimeIntegrator_DSTATE = 0.0;
  }

  /* Outputs for Atomic SubSystem: '<S343>/PID_Power' */
  Gen2_ref_DWork->DiscreteTimeIntegrator_PrevRese = (int8_T)
    rtb_LogicalOperator_in;

  /* End of Update for DiscreteIntegrator: '<S345>/Discrete-Time Integrator' */
  /* End of Outputs for SubSystem: '<S343>/PID_Power' */

  /* Update for Delay: '<S413>/Delay' */
  Gen2_ref_DWork->icLoad_n = false;
  Gen2_ref_DWork->Delay_DSTATE_n = rtb_Divide4_ia;

  /* Update for Delay: '<S881>/Delay' */
  Gen2_ref_DWork->icLoad_m = false;
  Gen2_ref_DWork->Delay_DSTATE_oh = rtb_Switch_ed;

  /* Update for Delay: '<S404>/Delay' */
  Gen2_ref_DWork->icLoad_k = false;
  Gen2_ref_DWork->Delay_DSTATE_g = rtb_Product_gj;

  /* Update for Delay: '<S15>/Resettable Delay' */
  Gen2_ref_DWork->icLoad_nl = false;
  Gen2_ref_DWork->ResettableDelay_DSTATE = Gen2_ref_B->Filter1_fj.Switch;

  /* Update for Delay: '<Root>/Delay4' */
  Gen2_ref_DWork->Delay4_DSTATE = rtb_TmpSignalConversionAtSFun_p[0];

  /* Update for Delay: '<Root>/Delay3' */
  Gen2_ref_DWork->Delay3_DSTATE = Gen2_ref_B->sf_IntegerZOH.y;

  /* Update for Delay: '<Root>/Delay6' incorporates:
   *  Logic: '<S18>/Logical Operator'
   *  Logic: '<S18>/Logical Operator1'
   *  Logic: '<S18>/Logical Operator3'
   *  Product: '<S18>/Divide'
   *  RelationalOperator: '<S18>/Relational Operator2'
   */
  Gen2_ref_DWork->Delay6_DSTATE = (((rtb_TmpSignalConversionAtSFun_p[0] /
    FILT_IN >= r) && rtb_bTV_sat) || (rtb_bCBV_min && rtb_bTV_sat));

  /* Update for Delay: '<Root>/Delay1' incorporates:
   *  SignalConversion generated from: '<Root>/Delay1'
   */
  Gen2_ref_DWork->Delay1_DSTATE[0] = rtb_Switch2_n5;
  Gen2_ref_DWork->Delay1_DSTATE[1] = rtb_Switch1_k;
  Gen2_ref_DWork->Delay1_DSTATE[2] = rtb_PactOut_o;

  /* Update for Delay: '<Root>/Delay2' */
  Gen2_ref_DWork->icLoad_e = false;
  Gen2_ref_DWork->Delay2_DSTATE = rtb_Product1_fu;

  /* Update for UnitDelay: '<S343>/Unit Delay1' */
  Gen2_ref_DWork->UnitDelay1_DSTATE = rtb_Switch_on;

  /* Update for UnitDelay: '<S343>/Unit Delay' incorporates:
   *  BusCreator: '<S389>/Bus Creator1'
   */
  Gen2_ref_DWork->UnitDelay_DSTATE_mg = rtb_BusCreator1_h_ui;

  /* Update for DiscreteIntegrator: '<S760>/Discrete-Time Integrator' incorporates:
   *  Logic: '<S743>/Logical Operator'
   */
  Gen2_ref_DWork->DiscreteTimeIntegrator_DSTATE_h += 0.01 * rtb_Divide_kp;
  if (Gen2_ref_DWork->DiscreteTimeIntegrator_DSTATE_h >= 1.0) {
    Gen2_ref_DWork->DiscreteTimeIntegrator_DSTATE_h = 1.0;
  } else if (Gen2_ref_DWork->DiscreteTimeIntegrator_DSTATE_h <= 0.0) {
    Gen2_ref_DWork->DiscreteTimeIntegrator_DSTATE_h = 0.0;
  }

  /* Outputs for Atomic SubSystem: '<S737>/Filter' */
  Gen2_ref_DWork->DiscreteTimeIntegrator_PrevRe_i = (int8_T)rtb_bResetHlci;

  /* End of Update for DiscreteIntegrator: '<S760>/Discrete-Time Integrator' */
  /* End of Outputs for SubSystem: '<S737>/Filter' */

  /* Update for Delay: '<S795>/Delay' */
  Gen2_ref_DWork->icLoad_h = false;
  Gen2_ref_DWork->Delay_DSTATE_b = rtb_Switch_jz;

  /* Update for UnitDelay: '<S761>/Unit Delay2' */
  Gen2_ref_DWork->UnitDelay2_DSTATE = rtb_rKK2_k;

  /* Update for DiscreteIntegrator: '<S579>/Discrete-Time Integrator' */
  Gen2_ref_DWork->DiscreteTimeIntegrator_DSTATE_m += 0.01 * rtb_Gain2_ao;

  /* Update for DiscreteIntegrator: '<S586>/Discrete-Time Integrator' */
  Gen2_ref_DWork->DiscreteTimeIntegrator_DSTATE_p += 0.01 * rtb_p2s;
  Gen2_ref_DWork->DiscreteTimeIntegrator_PrevRe_k = (int8_T)
    rtb_LogicalOperator1_j;

  /* Update for DiscreteIntegrator: '<S307>/Discrete-Time Integrator' */
  Gen2_ref_DWork->DiscreteTimeIntegrator_DSTATE_d += 0.01;
  if (Gen2_ref_DWork->DiscreteTimeIntegrator_DSTATE_d >= 1.0) {
    Gen2_ref_DWork->DiscreteTimeIntegrator_DSTATE_d = 1.0;
  } else if (Gen2_ref_DWork->DiscreteTimeIntegrator_DSTATE_d <= 0.0) {
    Gen2_ref_DWork->DiscreteTimeIntegrator_DSTATE_d = 0.0;
  }

  Gen2_ref_DWork->DiscreteTimeIntegrator_PrevRe_p = (int8_T)
    rtb_LogicalOperator2_e;

  /* End of Update for DiscreteIntegrator: '<S307>/Discrete-Time Integrator' */

  /* Update for UnitDelay: '<S14>/Unit Delay4' incorporates:
   *  Logic: '<Root>/Logical Operator'
   */
  Gen2_ref_DWork->UnitDelay4_DSTATE_d = rtb_LogicalOperator_cn;

  /* Update for Delay: '<S14>/Resettable Delay2' */
  Gen2_ref_DWork->icLoad_l = false;
  Gen2_ref_DWork->ResettableDelay2_DSTATE = rtb_Divide6_n;

  /* Update for Delay: '<S14>/Resettable Delay' */
  Gen2_ref_DWork->icLoad_i = false;
  Gen2_ref_DWork->ResettableDelay_DSTATE_l = Gen2_ref_B->Filter_l.Switch;

  /* Update for UnitDelay: '<S14>/Unit Delay' */
  Gen2_ref_DWork->UnitDelay_DSTATE = rtb_Product1_fu;

  /* Update for UnitDelay: '<S917>/Unit Delay' */
  Gen2_ref_DWork->UnitDelay_DSTATE_k = rtb_RelationalOperator_a;

  /* Update for DiscreteIntegrator: '<S917>/Discrete-Time Integrator' */
  Gen2_ref_DWork->DiscreteTimeIntegrator_DSTATE_c += 0.01;
  Gen2_ref_DWork->DiscreteTimeIntegrator_PrevR_ka = (int8_T)
    rtb_LogicalOperator_i;

  /* Update for Delay: '<S14>/Resettable Delay3' */
  Gen2_ref_DWork->icLoad_f = false;
  Gen2_ref_DWork->ResettableDelay3_DSTATE = rtb_RelationalOperator_l5;

  /* Update for UnitDelay: '<S641>/Unit Delay2' */
  Gen2_ref_DWork->UnitDelay2_DSTATE_d2 = rtb_LogicalOperator4_go;

  /* Update for DiscreteIntegrator: '<S748>/Discrete-Time Integrator' */
  Gen2_ref_DWork->DiscreteTimeIntegrator_IC_LOADI = 0U;
  Gen2_ref_DWork->DiscreteTimeIntegrator_DSTATE_k += 0.01 * rtb_MinMax_n;
  Gen2_ref_DWork->DiscreteTimeIntegrator_PrevRe_j = (int8_T)
    rtb_LogicalOperator1_e;

  /* Update for DiscreteIntegrator: '<S748>/Discrete-Time Integrator4' incorporates:
   *  DiscreteIntegrator: '<S748>/Discrete-Time Integrator'
   */
  Gen2_ref_DWork->DiscreteTimeIntegrator4_DSTATE += 0.01 * rtb_Divide3_d;
  if (Gen2_ref_DWork->DiscreteTimeIntegrator4_DSTATE >= 0.0) {
    Gen2_ref_DWork->DiscreteTimeIntegrator4_DSTATE = 0.0;
  } else if (Gen2_ref_DWork->DiscreteTimeIntegrator4_DSTATE <= -0.3) {
    Gen2_ref_DWork->DiscreteTimeIntegrator4_DSTATE = -0.3;
  }

  Gen2_ref_DWork->DiscreteTimeIntegrator4_PrevRes = (int8_T)
    rtb_LogicalOperator1_e;

  /* End of Update for DiscreteIntegrator: '<S748>/Discrete-Time Integrator4' */

  /* Update for DiscreteIntegrator: '<S748>/Discrete-Time Integrator1' incorporates:
   *  Sum: '<S748>/Sum2'
   */
  Gen2_ref_DWork->DiscreteTimeIntegrator1_DSTATE += (rtb_Product4_d +
    rtb_Divide2_f) * 0.01;
  Gen2_ref_DWork->DiscreteTimeIntegrator1_PrevRes = (int8_T)
    rtb_LogicalOperator3_fj;

  /* Update for Delay: '<S637>/Resettable Delay' */
  Gen2_ref_DWork->icLoad_ef = false;
  Gen2_ref_DWork->ResettableDelay_DSTATE_i = rtb_Sum2_kg;

  /* Update for Delay: '<S637>/Variable Integer Delay' */
  Gen2_ref_DWork->icLoad_b = false;
  Gen2_ref_DWork->VariableIntegerDelay_DSTATE[Gen2_ref_DWork->CircBufIdx] =
    rtb_Switch_jv;
  if (Gen2_ref_DWork->CircBufIdx < 199) {
    Gen2_ref_DWork->CircBufIdx++;
  } else {
    Gen2_ref_DWork->CircBufIdx = 0U;
  }

  /* End of Update for Delay: '<S637>/Variable Integer Delay' */

  /* Update for UnitDelay: '<S628>/Unit Delay1' */
  Gen2_ref_DWork->UnitDelay1_DSTATE_a = rtb_Product1_b4;

  /* Update for Delay: '<S625>/Delay' */
  Gen2_ref_DWork->Delay_DSTATE_k = rtb_kW2W;

  /* Update for Delay: '<S666>/Resettable Delay' */
  Gen2_ref_DWork->icLoad_i0 = false;
  for (i = 0; i < 13; i++) {
    Gen2_ref_DWork->ResettableDelay_DSTATE_a[i] =
      Gen2_ref_B->sf_MATLABFunction1_m.y_map_new[i];
  }

  /* End of Update for Delay: '<S666>/Resettable Delay' */

  /* Update for UnitDelay: '<S667>/Unit Delay2' */
  Gen2_ref_DWork->UnitDelay2_DSTATE_n = rtb_LogicalOperator4_go;

  /* Update for UnitDelay: '<S667>/Unit Delay1' */
  Gen2_ref_DWork->UnitDelay1_DSTATE_e = rtb_Divide3_g;

  /* Update for Delay: '<S714>/Resettable Delay1' */
  Gen2_ref_DWork->icLoad_np = false;

  /* Update for UnitDelay: '<S714>/Unit Delay1' */
  Gen2_ref_DWork->UnitDelay1_DSTATE_o = rtb_Switch2_au;

  /* Update for Delay: '<S714>/Resettable Delay' */
  Gen2_ref_DWork->icLoad_j = false;
  for (i = 0; i < 13; i++) {
    /* Update for Delay: '<S714>/Resettable Delay1' */
    Gen2_ref_DWork->ResettableDelay1_DSTATE[i] = rtb_ResettableDelay_br[i];

    /* Update for Delay: '<S714>/Resettable Delay' */
    Gen2_ref_DWork->ResettableDelay_DSTATE_m[i] = rtb_y_map_new_n[i];
  }

  /* Update for DiscreteIntegrator: '<S714>/Discrete-Time Integrator' incorporates:
   *  Logic: '<S714>/Logical Operator2'
   */
  Gen2_ref_DWork->DiscreteTimeIntegrator_DSTATE_l += 0.01 * rtb_Switch_ks;
  Gen2_ref_DWork->DiscreteTimeIntegrator_PrevRe_o = (int8_T)
    rtb_LogicalOperator2_k_tmp;

  /* Update for Delay: '<S715>/Resettable Delay1' */
  Gen2_ref_DWork->icLoad_a = false;

  /* Update for UnitDelay: '<S715>/Unit Delay1' */
  Gen2_ref_DWork->UnitDelay1_DSTATE_j = rtb_Switch3_le;

  /* Update for Delay: '<S715>/Resettable Delay' */
  Gen2_ref_DWork->icLoad_m3 = false;
  for (i = 0; i < 7; i++) {
    /* Update for Delay: '<S715>/Resettable Delay1' */
    Gen2_ref_DWork->ResettableDelay1_DSTATE_e[i] = rtb_Switch_dau[i];

    /* Update for Delay: '<S715>/Resettable Delay' */
    Gen2_ref_DWork->ResettableDelay_DSTATE_e[i] = rtb_y_map_new_a[i];
  }

  /* Update for DiscreteIntegrator: '<S715>/Discrete-Time Integrator' incorporates:
   *  Logic: '<S714>/Logical Operator2'
   */
  Gen2_ref_DWork->DiscreteTimeIntegrator_DSTATE_e += 0.01 * rtb_Divide2_a;
  Gen2_ref_DWork->DiscreteTimeIntegrator_PrevRe_n = (int8_T)
    rtb_LogicalOperator2_k_tmp;

  /* Update for DiscreteIntegrator: '<S748>/Discrete-Time Integrator3' incorporates:
   *  DiscreteIntegrator: '<S748>/Discrete-Time Integrator'
   */
  Gen2_ref_DWork->DiscreteTimeIntegrator3_DSTATE += 0.01 * rtb_Product1;
  Gen2_ref_DWork->DiscreteTimeIntegrator3_PrevRes = (int8_T)
    rtb_LogicalOperator1_e;

  /* Update for DiscreteIntegrator: '<S748>/Discrete-Time Integrator2' incorporates:
   *  DiscreteIntegrator: '<S748>/Discrete-Time Integrator'
   */
  Gen2_ref_DWork->DiscreteTimeIntegrator2_DSTATE += 0.01 * rtb_Pa2bar_k;
  Gen2_ref_DWork->DiscreteTimeIntegrator2_PrevRes = (int8_T)
    rtb_LogicalOperator1_e;

  /* Update for Delay: '<S431>/Delay' incorporates:
   *  SignalConversion generated from: '<S431>/Delay'
   */
  Gen2_ref_DWork->icLoad_b3 = false;
  Gen2_ref_DWork->Delay_DSTATE_ba[0] = rtb_Divide_ab[0];
  Gen2_ref_DWork->Delay_DSTATE_ba[1] = rtb_Divide_ab[1];
  Gen2_ref_DWork->Delay_DSTATE_ba[2] = rtb_Sum_c;
  Gen2_ref_DWork->Delay_DSTATE_ba[3] = rtb_Divide_ab[3];

  /* Update for UnitDelay: '<S606>/Unit Delay' */
  Gen2_ref_DWork->UnitDelay_DSTATE_ma = rtb_LogicalOperator1_ja;

  /* Update for Delay: '<S608>/Delay to avoid alg.loop' */
  Gen2_ref_DWork->Delaytoavoidalgloop_DSTATE = rtb_TOF_IN;

  /* Update for UnitDelay: '<S608>/Unit Delay' */
  Gen2_ref_DWork->TP_state = rtb_LogicalOperator1_pa;

  /* Update for UnitDelay: '<S611>/Delay Input1' */
  Gen2_ref_DWork->DelayInput1_DSTATE = rtb_LogicalOperator5;

  /* Update for DiscreteIntegrator: '<S608>/Discrete-Time Integrator' */
  Gen2_ref_DWork->DiscreteTimeIntegrator_DSTAT_h5 += 0.01 * rtb_Switch2_g3;
  Gen2_ref_DWork->DiscreteTimeIntegrator_PrevRe_m = (int8_T)
    rtb_LogicalOperator4_m5;

  /* Update for UnitDelay: '<S603>/Delay Input1' */
  Gen2_ref_DWork->DelayInput1_DSTATE_n = rtb_LogicalOperator1_pa;

  /* Update for UnitDelay: '<S581>/Unit Delay' */
  Gen2_ref_DWork->UnitDelay_DSTATE_f = rtb_Product1_aq;

  /* Update for UnitDelay: '<S716>/Unit Delay3' */
  Gen2_ref_DWork->UnitDelay3_DSTATE_go = Gen2_ref_B->TON_j.LogicalOperator3;

  /* Update for UnitDelay: '<S716>/Unit Delay2' */
  Gen2_ref_DWork->UnitDelay2_DSTATE_m = rtb_Switch1_cl[0];

  /* Update for UnitDelay: '<S716>/Unit Delay1' */
  for (i = 0; i < 13; i++) {
    Gen2_ref_DWork->UnitDelay1_DSTATE_f[i] = rtb_y_map_new[i];
  }

  /* End of Update for UnitDelay: '<S716>/Unit Delay1' */

  /* Update for UnitDelay: '<Root>/Unit Delay3' */
  Gen2_ref_DWork->UnitDelay3_DSTATE = rtb_TmpSignalConversionAtSFun_p[0];

  /* Update for UnitDelay: '<Root>/Unit Delay4' */
  Gen2_ref_DWork->UnitDelay4_DSTATE = Gen2_ref_B->sf_IntegerZOH.y;

  /* Update for UnitDelay: '<S1>/Unit Delay1' */
  Gen2_ref_DWork->UnitDelay1_DSTATE_ek = rtb_Switch1_kk;

  /* Update for UnitDelay: '<S31>/UD' */
  Gen2_ref_DWork->UD_DSTATE = rtb_LogicalOperator_hi;

  /* Update for UnitDelay: '<Root>/Unit Delay2' incorporates:
   *  Product: '<S5>/Divide2'
   *  Sum: '<S11>/Sum'
   *  Sum: '<S5>/Add2'
   */
  Gen2_ref_DWork->UnitDelay2_DSTATE_h[0] = rtb_Switch_fy_tmp_tmp * R_2inp[0] +
    rtb_Divide3_e[0];
  Gen2_ref_DWork->UnitDelay2_DSTATE_h[1] = rtb_Switch_fy_tmp_tmp * R_2inp[1] +
    rtb_Divide3_e[1];
  Gen2_ref_DWork->UnitDelay2_DSTATE_h[2] = rtb_Switch_fy_tmp_tmp * R_2inp[2] +
    rtb_Divide3_e[2];
  Gen2_ref_DWork->UnitDelay2_DSTATE_h[3] = rtb_Switch_fy_tmp_tmp * R_2inp[3] +
    rtb_Divide3_e[3];

  /* Update for UnitDelay: '<S62>/Unit Delay4' */
  Gen2_ref_DWork->UnitDelay4_DSTATE_k = Gen2_ref_B->TON_1.LogicalOperator3;

  /* Update for DiscreteIntegrator: '<S62>/Discrete-Time Integrator' */
  Gen2_ref_DWork->DiscreteTimeIntegrator_DSTATE_a += 0.01 * rtb_Gain_kl;
  if (Gen2_ref_DWork->DiscreteTimeIntegrator_DSTATE_a >= 1.0) {
    Gen2_ref_DWork->DiscreteTimeIntegrator_DSTATE_a = 1.0;
  } else if (Gen2_ref_DWork->DiscreteTimeIntegrator_DSTATE_a <= -0.1) {
    Gen2_ref_DWork->DiscreteTimeIntegrator_DSTATE_a = -0.1;
  }

  Gen2_ref_DWork->DiscreteTimeIntegrator_PrevR_oa = (int8_T)
    rtb_LogicalOperator1_i2;

  /* End of Update for DiscreteIntegrator: '<S62>/Discrete-Time Integrator' */

  /* Update for Delay: '<S78>/Variable Integer Delay' */
  Gen2_ref_DWork->icLoad_ev = false;

  /* Update for UnitDelay: '<S78>/Unit Delay' */
  Gen2_ref_DWork->UnitDelay_DSTATE_e = rtb_p1LP;

  /* Update for Delay: '<S88>/Delay' */
  Gen2_ref_DWork->icLoad_d = false;
  Gen2_ref_DWork->Delay_DSTATE_ko = rtb_p2HP;

  /* Update for Delay: '<S90>/Delay' */
  Gen2_ref_DWork->icLoad_es = false;
  Gen2_ref_DWork->Delay_DSTATE_j = rtb_Sum4_g;

  /* Update for Delay: '<S87>/Delay' */
  Gen2_ref_DWork->icLoad_evr = false;
  Gen2_ref_DWork->Delay_DSTATE_m = rtb_Sum5_iu;

  /* Update for Delay: '<S89>/Delay' */
  Gen2_ref_DWork->icLoad_fg = false;
  Gen2_ref_DWork->Delay_DSTATE_d = rtb_Switch9_k;

  /* Update for Delay: '<S77>/Variable Integer Delay' */
  Gen2_ref_DWork->icLoad_c = false;
  for (k = 0; k < 299; k++) {
    /* Update for Delay: '<S78>/Variable Integer Delay' */
    Gen2_ref_DWork->VariableIntegerDelay_DSTATE_b[k] =
      Gen2_ref_DWork->VariableIntegerDelay_DSTATE_b[k + 1];

    /* Update for Delay: '<S77>/Variable Integer Delay' */
    Gen2_ref_DWork->VariableIntegerDelay_DSTATE_e[k] =
      Gen2_ref_DWork->VariableIntegerDelay_DSTATE_e[k + 1];
  }

  /* Update for Delay: '<S78>/Variable Integer Delay' */
  Gen2_ref_DWork->VariableIntegerDelay_DSTATE_b[299] = rtb_p1HP;

  /* Update for Delay: '<S77>/Variable Integer Delay' */
  Gen2_ref_DWork->VariableIntegerDelay_DSTATE_e[299] = rtb_p1HP;

  /* Update for UnitDelay: '<S77>/Unit Delay' */
  Gen2_ref_DWork->UnitDelay_DSTATE_d = rtb_Sum3_o;

  /* Update for Delay: '<S80>/Delay' */
  Gen2_ref_DWork->icLoad_eu = false;
  Gen2_ref_DWork->Delay_DSTATE_g2 = rtb_Switch_czo;

  /* Update for Delay: '<S82>/Delay' */
  Gen2_ref_DWork->icLoad_ee = false;
  Gen2_ref_DWork->Delay_DSTATE_dm = rtb_UkYk1_a4;

  /* Update for Delay: '<S79>/Delay' */
  Gen2_ref_DWork->icLoad_ki = false;
  Gen2_ref_DWork->Delay_DSTATE_jl = rtb_Gain_i;

  /* Update for Delay: '<S81>/Delay' */
  Gen2_ref_DWork->icLoad_h3 = false;
  Gen2_ref_DWork->Delay_DSTATE_h = rtb_Saturation_e;

  /* Update for Delay: '<S23>/Delay' */
  Gen2_ref_DWork->Delay_DSTATE_lv = rtb_LogicalOperator;

  /* Update for UnitDelay: '<S53>/Unit Delay4' */
  Gen2_ref_DWork->UnitDelay4_DSTATE_o = rtb_LogicalOperator2_p1;

  /* Update for Delay: '<S63>/Delay' */
  Gen2_ref_DWork->icLoad_g = false;
  Gen2_ref_DWork->Delay_DSTATE_c = rtb_deltafalllimit_h0;

  /* Update for Delay: '<S64>/Delay' */
  Gen2_ref_DWork->icLoad_c1 = false;
  Gen2_ref_DWork->Delay_DSTATE_i = rtb_Switch1_lk;

  /* Update for DiscreteIntegrator: '<S48>/Discrete-Time Integrator' */
  Gen2_ref_DWork->DiscreteTimeIntegrator_DSTAT_ac += 0.01 * rtb_Switch_eu;
  if (Gen2_ref_DWork->DiscreteTimeIntegrator_DSTAT_ac >= 1.0) {
    Gen2_ref_DWork->DiscreteTimeIntegrator_DSTAT_ac = 1.0;
  } else if (Gen2_ref_DWork->DiscreteTimeIntegrator_DSTAT_ac <= 0.0) {
    Gen2_ref_DWork->DiscreteTimeIntegrator_DSTAT_ac = 0.0;
  }

  Gen2_ref_DWork->DiscreteTimeIntegrator_PrevRe_l = (int8_T)
    rtb_LogicalOperator2_dc;

  /* Update for UnitDelay: '<S23>/Unit Delay3' */
  Gen2_ref_DWork->UnitDelay3_DSTATE_gf = rtb_LogicalOperator2_dc;

  /* Update for UnitDelay: '<S427>/Unit Delay1' */
  Gen2_ref_DWork->UnitDelay1_DSTATE_m = rtb_LogicalOperator1_a0;

  /* Update for DiscreteIntegrator: '<S132>/Discrete-Time Integrator' */
  Gen2_ref_DWork->DiscreteTimeIntegrator_DSTATE_g += 0.01 * rtb_Gain1_fr;

  /* Update for UnitDelay: '<S160>/Delay Input1' */
  Gen2_ref_DWork->DelayInput1_DSTATE_f = Gen2_ref_B->BusInput3.bdcTv.bActive_ff;

  /* Update for UnitDelay: '<S45>/Unit Delay1' */
  Gen2_ref_DWork->UnitDelay1_DSTATE_ed = rtb_Product1_bc;

  /* Update for Delay: '<S45>/Delay' */
  Gen2_ref_DWork->icLoad_eh = false;
  Gen2_ref_DWork->Delay_DSTATE_cn =
    Gen2_ref_B->Inverse_Linearization1.LCRScal_Lam_EOT1;

  /* Update for Delay: '<S161>/Delay2' */
  Gen2_ref_DWork->Delay2_DSTATE_f = rtb_LogicalOperator3_k;

  /* Update for Delay: '<S161>/Delay1' */
  Gen2_ref_DWork->Delay1_DSTATE_l = rtb_Sum8_m;

  /* Update for Delay: '<S161>/Delay' */
  Gen2_ref_DWork->Delay_DSTATE_gp = rtb_Product1_bc;

  /* Update for DiscreteIntegrator: '<S45>/Discrete-Time Integrator1' incorporates:
   *  MATLAB Function: '<S45>/tv_fb_err'
   *  Product: '<S45>/Product1'
   *  Sum: '<S45>/Sum3'
   */
  Gen2_ref_DWork->DiscreteTimeIntegrator1_IC_LOAD = 0U;
  Gen2_ref_DWork->DiscreteTimeIntegrator1_DSTAT_n += (rtb_Sum10 * rtb_Switch2_j0
    + rtb_Switch2_oou) * 0.01;
  Gen2_ref_DWork->DiscreteTimeIntegrator1_PrevR_k = (int8_T)
    rtb_LogicalOperator3_aa;

  /* Update for UnitDelay: '<S41>/Unit Delay' */
  Gen2_ref_DWork->UnitDelay_DSTATE_je = rtb_Switch4_j;

  /* Update for UnitDelay: '<S1>/Unit Delay5' */
  Gen2_ref_DWork->UnitDelay5_DSTATE = rtb_Switch1_kk;

  /* Update for UnitDelay: '<S1>/Unit Delay' */
  Gen2_ref_DWork->UnitDelay_DSTATE_i = rtb_Switch13;

  /* Update for DiscreteIntegrator: '<S133>/Discrete-Time Integrator' */
  Gen2_ref_DWork->DiscreteTimeIntegrator_DSTATE_j += 0.01 * rtb_Saturation;
  Gen2_ref_DWork->DiscreteTimeIntegrator_PrevR_no = (int8_T)
    rtb_LogicalOperator1_ix;

  /* Update for UnitDelay: '<S27>/Unit Delay6' */
  Gen2_ref_DWork->UnitDelay6_DSTATE = rtb_Sum1_lo;

  /* Update for UnitDelay: '<S107>/Delay Input1' */
  Gen2_ref_DWork->DelayInput1_DSTATE_fv =
    Gen2_ref_B->BusInput3.bdcCbv.bActive_ff;

  /* Update for UnitDelay: '<S26>/Unit Delay1' */
  Gen2_ref_DWork->UnitDelay1_DSTATE_c = rtb_MultiportSwitch;

  /* Update for Delay: '<S26>/Delay' */
  Gen2_ref_DWork->icLoad_kq = false;
  Gen2_ref_DWork->Delay_DSTATE_hq = rtb_Saturation1_i;

  /* Update for Delay: '<S111>/Delay2' */
  Gen2_ref_DWork->Delay2_DSTATE_k = rtb_LogicalOperator5_p;

  /* Update for Delay: '<S111>/Delay' */
  Gen2_ref_DWork->Delay_DSTATE_ow = rtb_MultiportSwitch;

  /* Update for DiscreteIntegrator: '<S26>/Discrete-Time Integrator' */
  Gen2_ref_DWork->DiscreteTimeIntegrator_IC_LOA_l = 0U;
  Gen2_ref_DWork->DiscreteTimeIntegrator_DSTAT_ja += 0.01 * rtb_Switch1_mm;
  Gen2_ref_DWork->DiscreteTimeIntegrator_PrevRe_c = (int8_T)
    rtb_LogicalOperator_b;

  /* Update for UnitDelay: '<S1>/Unit Delay2' */
  Gen2_ref_DWork->UnitDelay2_DSTATE_d = rtb_Switch1_kk;

  /* Update for UnitDelay: '<S1>/Unit Delay3' */
  Gen2_ref_DWork->UnitDelay3_DSTATE_g = rtb_Switch1_kk;

  /* Update for UnitDelay: '<S46>/Unit Delay' */
  Gen2_ref_DWork->UnitDelay_DSTATE_b = rtb_Switch2_by;

  /* Update for UnitDelay: '<S491>/Unit Delay2' */
  Gen2_ref_DWork->UnitDelay2_DSTATE_j = rtb_LogicalOperator_aw;

  /* Update for Delay: '<S494>/Delay' */
  Gen2_ref_DWork->icLoad_ir = false;
  Gen2_ref_DWork->Delay_DSTATE_f = rtb_Switch2_l;

  /* Update for DiscreteIntegrator: '<S22>/Discrete-Time Integrator' incorporates:
   *  DiscreteIntegrator: '<S48>/Discrete-Time Integrator'
   *  Sum: '<S22>/Sum2'
   */
  Gen2_ref_DWork->DiscreteTimeIntegrator_DSTATE_i += (delta_y - rtb_Gain) * 0.01;
  if (Gen2_ref_DWork->DiscreteTimeIntegrator_DSTATE_i >= 1.0) {
    Gen2_ref_DWork->DiscreteTimeIntegrator_DSTATE_i = 1.0;
  } else if (Gen2_ref_DWork->DiscreteTimeIntegrator_DSTATE_i <= 0.0) {
    Gen2_ref_DWork->DiscreteTimeIntegrator_DSTATE_i = 0.0;
  }

  Gen2_ref_DWork->DiscreteTimeIntegrator_PrevR_jc = (int8_T)
    rtb_LogicalOperator2_dc;

  /* End of Update for DiscreteIntegrator: '<S22>/Discrete-Time Integrator' */

  /* Update for UnitDelay: '<S427>/Unit Delay5' */
  Gen2_ref_DWork->TOF_2_state = Gen2_ref_B->TOF2_d.LogicalOperator1;

  /* Update for UnitDelay: '<S427>/Unit Delay3' */
  Gen2_ref_DWork->UnitDelay3_DSTATE_h5 =
    Gen2_ref_B->TP_Misfire_ON_2ndtime.LogicalOperator1;

  /* Update for UnitDelay: '<S427>/Unit Delay2' */
  Gen2_ref_DWork->UnitDelay2_DSTATE_hh = rtb_dbg_HLCi;

  /* Update for UnitDelay: '<S634>/Unit Delay' */
  Gen2_ref_DWork->UnitDelay_DSTATE_kx = rtb_LogicalOperator5_mv;

  /* Update for Delay: '<S708>/Delay' */
  Gen2_ref_DWork->icLoad_nv = false;
  Gen2_ref_DWork->Delay_DSTATE_l = rtb_Divide5_h;

  /* Update for UnitDelay: '<S427>/Unit Delay6' */
  Gen2_ref_DWork->UnitDelay6_DSTATE_m = rtb_Divide4_d;

  /* Update for UnitDelay: '<S427>/Unit Delay' */
  Gen2_ref_DWork->UnitDelay_DSTATE_n = rtb_RelationalOperator2_j;

  /* Update for Delay: '<S524>/Delay' */
  Gen2_ref_DWork->icLoad_dk = false;
  Gen2_ref_DWork->Delay_DSTATE_p = rtb_Switch5_iq;

  /* Update for Delay: '<S811>/Delay' */
  Gen2_ref_DWork->icLoad_iv = false;
  Gen2_ref_DWork->Delay_DSTATE_i4 = rtb_Sum4_ny;

  /* Update for Delay: '<S830>/Resettable Delay' */
  Gen2_ref_DWork->icLoad_ix = false;
  for (i = 0; i < 13; i++) {
    Gen2_ref_DWork->ResettableDelay_DSTATE_k[i] =
      Gen2_ref_B->sf_MATLABFunction1_l.y_map_new[i];
  }

  /* End of Update for Delay: '<S830>/Resettable Delay' */

  /* Update for UnitDelay: '<S831>/Unit Delay2' */
  Gen2_ref_DWork->UnitDelay2_DSTATE_i = rtb_LogicalOperator2_fy;

  /* Update for UnitDelay: '<S831>/Unit Delay1' incorporates:
   *  Constant: '<S12>/Constant'
   */
  Gen2_ref_DWork->UnitDelay1_DSTATE_n = 0.0;

  /* Update for Delay: '<S830>/Delay' */
  Gen2_ref_DWork->Delay_DSTATE_n2 = rtb_LogicalOperator2_l;

  /* Update for Delay: '<S666>/Delay' */
  Gen2_ref_DWork->Delay_DSTATE_cnq = rtb_LogicalOperator_f;

  /* Update for UnitDelay: '<S635>/Unit Delay1' */
  Gen2_ref_DWork->UnitDelay1_DSTATE_eq = rtb_kW2W1_h;

  /* Update for UnitDelay: '<S635>/Unit Delay2' */
  Gen2_ref_DWork->UnitDelay2_DSTATE_di = rtb_Gain6_b;

  /* Update for Delay: '<S714>/Delay' incorporates:
   *  Logic: '<S714>/Logical Operator2'
   */
  Gen2_ref_DWork->Delay_DSTATE_a = rtb_LogicalOperator2_k_tmp;

  /* Update for Delay: '<S715>/Delay' */
  Gen2_ref_DWork->Delay_DSTATE_ng = rtb_LogicalOperator2_k_tmp;

  /* Update for UnitDelay: '<S275>/Unit Delay' */
  Gen2_ref_DWork->UnitDelay_DSTATE_dk = rtb_SumofElements;

  /* Update for UnitDelay: '<S275>/Unit Delay1' */
  Gen2_ref_DWork->UnitDelay1_DSTATE_b = rtb_Gain6_jx;

  /* Update for UnitDelay: '<S275>/Unit Delay2' */
  Gen2_ref_DWork->UnitDelay2_DSTATE_k = rtb_SumofElements;

  /* Update for UnitDelay: '<S275>/Unit Delay3' */
  Gen2_ref_DWork->UnitDelay3_DSTATE_m = rtb_Gain7;

  /* Update for UnitDelay: '<S291>/Unit Delay' */
  Gen2_ref_DWork->UnitDelay_DSTATE_m = rtb_SumofElements_l;

  /* Update for UnitDelay: '<S291>/Unit Delay1' */
  Gen2_ref_DWork->UnitDelay1_DSTATE_c2 = rtb_Sum_ig;

  /* Update for UnitDelay: '<S291>/Unit Delay2' */
  Gen2_ref_DWork->UnitDelay2_DSTATE_p = rtb_SumofElements_l;

  /* Update for UnitDelay: '<S291>/Unit Delay3' */
  Gen2_ref_DWork->UnitDelay3_DSTATE_h = rtb_Sum_gb;

  /* Update for UnitDelay: '<S133>/Unit Delay' */
  Gen2_ref_DWork->UnitDelay_DSTATE_o = rtb_RelationalOperator1_j;

  /* Update for UnitDelay: '<S15>/Unit Delay' */
  Gen2_ref_DWork->UnitDelay_DSTATE_fm = rtb_mbar2pa_g;

  /* Update for UnitDelay: '<S10>/Unit Delay' */
  Gen2_ref_DWork->UnitDelay_DSTATE_j = 4140004U;
}

/* Model initialize function */
void Gen2_ref_initialize(RT_MODEL_Gen2_ref *const Gen2_ref_M, struct Gen2* inst)
{
  struct D_Work_Gen2_ref *Gen2_ref_DWork = Gen2_ref_M->dwork;
  struct PrevZCSigStates_Gen2_ref *Gen2_ref_PrevZCSigState = Gen2_ref_M->prevZCSigState;

  /* Registration code */

  /* initialize non-finites */
  rt_InitInfAndNaN(sizeof(real_T));
  Gen2_ref_PrevZCSigState->Delay_Reset_ZCE = UNINITIALIZED_ZCSIG;
  Gen2_ref_PrevZCSigState->Delay_Reset_ZCE_k = UNINITIALIZED_ZCSIG;
  Gen2_ref_PrevZCSigState->Delay_Reset_ZCE_b = UNINITIALIZED_ZCSIG;
  Gen2_ref_PrevZCSigState->Delay_Reset_ZCE_n = UNINITIALIZED_ZCSIG;
  Gen2_ref_PrevZCSigState->ResettableDelay_Reset_ZCE = UNINITIALIZED_ZCSIG;
  Gen2_ref_PrevZCSigState->Delay2_Reset_ZCE = UNINITIALIZED_ZCSIG;
  Gen2_ref_PrevZCSigState->Delay_Reset_ZCE_m = UNINITIALIZED_ZCSIG;
  Gen2_ref_PrevZCSigState->ResettableDelay_Reset_ZCE_j = UNINITIALIZED_ZCSIG;
  Gen2_ref_PrevZCSigState->ResettableDelay3_Reset_ZCE = UNINITIALIZED_ZCSIG;
  Gen2_ref_PrevZCSigState->ResettableDelay_Reset_ZCE_m = UNINITIALIZED_ZCSIG;
  Gen2_ref_PrevZCSigState->VariableIntegerDelay_Reset_ZCE = UNINITIALIZED_ZCSIG;
  Gen2_ref_PrevZCSigState->ResettableDelay_Reset_ZCE_a = POS_ZCSIG;
  Gen2_ref_PrevZCSigState->ResettableDelay1_Reset_ZCE = POS_ZCSIG;
  Gen2_ref_PrevZCSigState->ResettableDelay_Reset_ZCE_e = POS_ZCSIG;
  Gen2_ref_PrevZCSigState->ResettableDelay1_Reset_ZCE_g = POS_ZCSIG;
  Gen2_ref_PrevZCSigState->ResettableDelay_Reset_ZCE_b = POS_ZCSIG;
  Gen2_ref_PrevZCSigState->VariableIntegerDelay_Reset_ZC_i = UNINITIALIZED_ZCSIG;
  Gen2_ref_PrevZCSigState->Delay_Reset_ZCE_d = UNINITIALIZED_ZCSIG;
  Gen2_ref_PrevZCSigState->Delay_Reset_ZCE_l = UNINITIALIZED_ZCSIG;
  Gen2_ref_PrevZCSigState->Delay_Reset_ZCE_i = UNINITIALIZED_ZCSIG;
  Gen2_ref_PrevZCSigState->Delay_Reset_ZCE_mu = UNINITIALIZED_ZCSIG;
  Gen2_ref_PrevZCSigState->VariableIntegerDelay_Reset_ZC_o = UNINITIALIZED_ZCSIG;
  Gen2_ref_PrevZCSigState->Delay_Reset_ZCE_d3 = UNINITIALIZED_ZCSIG;
  Gen2_ref_PrevZCSigState->Delay_Reset_ZCE_c = UNINITIALIZED_ZCSIG;
  Gen2_ref_PrevZCSigState->Delay_Reset_ZCE_p = UNINITIALIZED_ZCSIG;
  Gen2_ref_PrevZCSigState->Delay_Reset_ZCE_ih = UNINITIALIZED_ZCSIG;
  Gen2_ref_PrevZCSigState->Delay_Reset_ZCE_k2 = UNINITIALIZED_ZCSIG;
  Gen2_ref_PrevZCSigState->Delay_Reset_ZCE_a = UNINITIALIZED_ZCSIG;
  Gen2_ref_PrevZCSigState->Delay_Reset_ZCE_o = UNINITIALIZED_ZCSIG;
  Gen2_ref_PrevZCSigState->Delay_Reset_ZCE_kk = UNINITIALIZED_ZCSIG;
  Gen2_ref_PrevZCSigState->Delay_Reset_ZCE_bc = UNINITIALIZED_ZCSIG;
  Gen2_ref_PrevZCSigState->Delay_Reset_ZCE_j = UNINITIALIZED_ZCSIG;
  Gen2_ref_PrevZCSigState->Delay_Reset_ZCE_h = UNINITIALIZED_ZCSIG;
  Gen2_ref_PrevZCSigState->Delay_Reset_ZCE_bi = UNINITIALIZED_ZCSIG;
  Gen2_ref_PrevZCSigState->ResettableDelay_Reset_ZCE_k = POS_ZCSIG;
  Gen2_ref_PrevZCSigState->Delay_Reset_ZCE_at = UNINITIALIZED_ZCSIG;
  Gen2_ref_PrevZCSigState->Delay_Reset_ZCE_e = UNINITIALIZED_ZCSIG;
  Gen2_ref_PrevZCSigState->Delay_Reset_ZCE_mt = UNINITIALIZED_ZCSIG;

  /* InitializeConditions for Delay: '<S425>/Delay' */
  Gen2_ref_DWork->icLoad = true;

  /* InitializeConditions for DiscreteIntegrator: '<S345>/Discrete-Time Integrator' */
  Gen2_ref_DWork->DiscreteTimeIntegrator_DSTATE = 1.0;

  /* InitializeConditions for Delay: '<S413>/Delay' */
  Gen2_ref_DWork->icLoad_n = true;

  /* InitializeConditions for Delay: '<S881>/Delay' */
  Gen2_ref_DWork->icLoad_m = true;

  /* InitializeConditions for Delay: '<S404>/Delay' */
  Gen2_ref_DWork->icLoad_k = true;
```
